LIN {X 0,Y 217.239,Z 668.067,A -85,B 0,C 180,E1 -28167.228,E2 -28167.228} C_VEL
LIN {X 0,Y 217.016,Z 676.061,A -85,B 0,C 180,E1 -28170,E2 -28170} C_VEL
LIN {X 0,Y 216.714,Z 682.608,A -85,B 0,C 180,E1 -28172.779,E2 -28172.779} C_VEL
LIN {X 0,Y 216.451,Z 688.034,A -85,B 0,C 180,E1 -28175.571,E2 -28175.571} C_VEL
LIN {X 0,Y 216.7,Z 693.898,A -85,B 0,C 180,E1 -28179.3,E2 -28179.3} C_VEL
LIN {X 0,Y 217.929,Z 698.427,A -85,B 0,C 180,E1 -28183.002,E2 -28183.002} C_VEL
LIN {X 0,Y 220.325,Z 701.768,A -85,B 0,C 180,E1 -28186.626,E2 -28186.626} C_VEL
LIN {X 0,Y 224.003,Z 703.996,A -85,B 0,C 180,E1 -28190.118,E2 -28190.118} C_VEL
LIN {X 0,Y 228.64,Z 705.109,A -85,B 0,C 180,E1 -28193.469,E2 -28193.469} C_VEL
LIN {X 0,Y 234.186,Z 705.102,A -85,B 0,C 180,E1 -28196.657,E2 -28196.657} C_VEL
LIN {X 0,Y 240.893,Z 703.976,A -85,B 0,C 180,E1 -28199.624,E2 -28199.624} C_VEL
LIN {X 0,Y 248.473,Z 701.716,A -85,B 0,C 180,E1 -28202.385,E2 -28202.385} C_VEL
LIN {X 0,Y 256.781,Z 698.288,A -85,B 0,C 180,E1 -28204.948,E2 -28204.948} C_VEL
LIN {X 0,Y 265.851,Z 693.598,A -85,B 0,C 180,E1 -28207.3,E2 -28207.3} C_VEL
LIN {X 0,Y 275.55,Z 687.57,A -85,B 0,C 180,E1 -28209.457,E2 -28209.457} C_VEL
LIN {X 0,Y 285.928,Z 680.01,A -85,B 0,C 180,E1 -28211.409,E2 -28211.409} C_VEL
LIN {X 0,Y 295.434,Z 671.975,A -85,B 0,C 180,E1 -28212.971,E2 -28212.971} C_VEL
LIN {X 0,Y 305.558,Z 662.13,A -85,B 0,C 180,E1 -28214.425,E2 -28214.425} C_VEL
LIN {X 0,Y 309.138,Z 658.314,A -85,B 0,C 180,E1 -28214.894,E2 -28214.894} C_VEL
LIN {X 0,Y 308.469,Z 659.033,A -85,B 0,C 180,E1 -28215.258,E2 -28215.258} C_VEL
LIN {X 0,Y 298.953,Z 668.646,A -85,B 0,C 180,E1 -28216.579,E2 -28216.579} C_VEL
LIN {X 0,Y 288.846,Z 677.542,A -85,B 0,C 180,E1 -28218.174,E2 -28218.174} C_VEL
LIN {X 0,Y 278.403,Z 685.481,A -85,B 0,C 180,E1 -28220.092,E2 -28220.092} C_VEL
LIN {X 0,Y 268.541,Z 691.868,A -85,B 0,C 180,E1 -28222.197,E2 -28222.197} C_VEL
LIN {X 0,Y 259.322,Z 696.857,A -85,B 0,C 180,E1 -28224.499,E2 -28224.499} C_VEL
LIN {X 0,Y 252.853,Z 699.744,A -85,B 0,C 180,E1 -28226.356,E2 -28226.356} C_VEL
LIN {X 0,Y 244.939,Z 702.551,A -85,B 0,C 180,E1 -28229.02,E2 -28229.02} C_VEL
LIN {X 0,Y 237.854,Z 704.212,A -85,B 0,C 180,E1 -28231.89,E2 -28231.89} C_VEL
LIN {X 0,Y 231.589,Z 704.754,A -85,B 0,C 180,E1 -28234.949,E2 -28234.949} C_VEL
LIN {X 0,Y 226.489,Z 704.166,A -85,B 0,C 180,E1 -28238.216,E2 -28238.216} C_VEL
LIN {X 0,Y 222.289,Z 702.473,A -85,B 0,C 180,E1 -28241.633,E2 -28241.633} C_VEL
LIN {X 0,Y 219.173,Z 699.666,A -85,B 0,C 180,E1 -28245.187,E2 -28245.187} C_VEL
LIN {X 0,Y 217.112,Z 695.687,A -85,B 0,C 180,E1 -28248.839,E2 -28248.839} C_VEL
LIN {X 0,Y 216.411,Z 690.516,A -85,B 0,C 180,E1 -28252.562,E2 -28252.562} C_VEL
LIN {X 0,Y 216.378,Z 683.877,A -85,B 0,C 180,E1 -28256.288,E2 -28256.288} C_VEL
LIN {X 0,Y 216.81,Z 676.605,A -85,B 0,C 180,E1 -28259.538,E2 -28259.538} C_VEL
LIN {X 0,Y 217.071,Z 668.937,A -85,B 0,C 180,E1 -28262.312,E2 -28262.312} C_VEL
LIN {X 0,Y 217.177,Z 661.275,A -85,B 0,C 180,E1 -28264.625,E2 -28264.625} C_VEL
LIN {X 0,Y 217.564,Z 649.405,A -85,B 0,C 180,E1 -28267.632,E2 -28267.632} C_VEL
LIN {X 0,Y 218.06,Z 637.025,A -85,B 0,C 180,E1 -28270.176,E2 -28270.176} C_VEL
LIN {X 0,Y 218.634,Z 624.743,A -85,B 0,C 180,E1 -28272.255,E2 -28272.255} C_VEL
LIN {X 0,Y 219.439,Z 609.747,A -85,B 0,C 180,E1 -28274.323,E2 -28274.323} C_VEL
LIN {X 0,Y 220.122,Z 596.007,A -85,B 0,C 180,E1 -28275.812,E2 -28275.812} C_VEL
LIN {X 0,Y 220.726,Z 579.884,A -85,B 0,C 180,E1 -28277.129,E2 -28277.129} C_VEL
LIN {X 0,Y 222.344,Z 529.839,A -85,B 0,C 180,E1 -28280.216,E2 -28280.216} C_VEL
LIN {X 0,Y 224.364,Z 480.881,A -85,B 0,C 180,E1 -28283.122,E2 -28283.122} C_VEL
LIN {X 0,Y 222.412,Z 452.386,A -85,B 0,C 180,E1 -28284.782,E2 -28284.782} C_VEL
LIN {X 0,Y 222.243,Z 439.496,A -85,B 0,C 180,E1 -28285.563,E2 -28285.563} C_VEL
LIN {X 0,Y 225.384,Z 413.949,A -85,B 0,C 180,E1 -28290.85,E2 -28290.85} C_VEL
LIN {X 0,Y 226.091,Z 408.23,A -85,B 0,C 180,E1 -28292.026,E2 -28292.026} C_VEL
LIN {X 0,Y 221.954,Z 389.076,A -85,B 0,C 180,E1 -28296.281,E2 -28296.281} C_VEL
LIN {X 0,Y 217.974,Z 370.88,A -85,B 0,C 180,E1 -28300.539,E2 -28300.539} C_VEL
LIN {X 0,Y 217.957,Z 370.883,A -85,B 0,C 180,E1 -28305.008,E2 -28305.008} C_VEL
LIN {X 0,Y 217.914,Z 370.887,A -85,B 0,C 180,E1 -28309.995,E2 -28309.995} C_VEL
LIN {X 0,Y 217.915,Z 371.065,A -85,B 0,C 180,E1 -28312.499,E2 -28312.499} C_VEL
LIN {X 0,Y 218.846,Z 373.704,A -85,B 0,C 180,E1 -28312.823,E2 -28312.823} C_VEL
LIN {X 0,Y 220.752,Z 376.135,A -85,B 0,C 180,E1 -28313.348,E2 -28313.348} C_VEL
LIN {X 0,Y 228.182,Z 388.008,A -85,B 0,C 180,E1 -28315.37,E2 -28315.37} C_VEL
LIN {X 0,Y 235.262,Z 400.411,A -85,B 0,C 180,E1 -28317.173,E2 -28317.173} C_VEL
LIN {X 0,Y 242.271,Z 414.273,A -85,B 0,C 180,E1 -28318.874,E2 -28318.874} C_VEL
LIN {X 0,Y 245.306,Z 421.27,A -85,B 0,C 180,E1 -28319.604,E2 -28319.604} C_VEL
LIN {X 0,Y 243.354,Z 467.862,A -85,B 0,C 180,E1 -28320.91,E2 -28320.91} C_VEL
LIN {X 0,Y 242.688,Z 488.569,A -85,B 0,C 180,E1 -28321.593,E2 -28321.593} C_VEL
LIN {X 0,Y 241.708,Z 502.885,A -85,B 0,C 180,E1 -28322.376,E2 -28322.376} C_VEL
LIN {X 0,Y 240.063,Z 516.937,A -85,B 0,C 180,E1 -28323.463,E2 -28323.463} C_VEL
LIN {X 0,Y 238.085,Z 529.464,A -85,B 0,C 180,E1 -28324.749,E2 -28324.749} C_VEL
LIN {X 0,Y 235.873,Z 541.665,A -85,B 0,C 180,E1 -28326.366,E2 -28326.366} C_VEL
LIN {X 0,Y 233.439,Z 552.842,A -85,B 0,C 180,E1 -28328.203,E2 -28328.203} C_VEL
LIN {X 0,Y 230.488,Z 564.111,A -85,B 0,C 180,E1 -28330.471,E2 -28330.471} C_VEL
LIN {X 0,Y 227.585,Z 574.185,A -85,B 0,C 180,E1 -28332.999,E2 -28332.999} C_VEL
LIN {X 0,Y 225.054,Z 582.522,A -85,B 0,C 180,E1 -28335.583,E2 -28335.583} C_VEL
LIN {X 0,Y 222.582,Z 590.486,A -85,B 0,C 180,E1 -28338.657,E2 -28338.657} C_VEL
LIN {X 0,Y 220.534,Z 596.925,A -85,B 0,C 180,E1 -28341.783,E2 -28341.783} C_VEL
LIN {X 0,Y 218.897,Z 602.636,A -85,B 0,C 180,E1 -28345.412,E2 -28345.412} C_VEL
LIN {X 0,Y 217.896,Z 605.963,A -85,B 0,C 180,E1 -28348.158,E2 -28348.158} C_VEL
LIN {X 0,Y 217.342,Z 609.076,A -85,B 0,C 180,E1 -28351.847,E2 -28351.847} C_VEL
LIN {X 0,Y 217.4,Z 610.861,A -85,B 0,C 180,E1 -28355.547,E2 -28355.547} C_VEL
LIN {X 0,Y 217.897,Z 611.372,A -85,B 0,C 180,E1 -28359.25,E2 -28359.25} C_VEL
LIN {X 0,Y 218.987,Z 610.594,A -85,B 0,C 180,E1 -28362.939,E2 -28362.939} C_VEL
LIN {X 0,Y 220.846,Z 608.486,A -85,B 0,C 180,E1 -28366.586,E2 -28366.586} C_VEL
LIN {X 0,Y 223.353,Z 604.998,A -85,B 0,C 180,E1 -28370.18,E2 -28370.18} C_VEL
LIN {X 0,Y 226.54,Z 600.015,A -85,B 0,C 180,E1 -28373.701,E2 -28373.701} C_VEL
LIN {X 0,Y 229.333,Z 595.158,A -85,B 0,C 180,E1 -28376.287,E2 -28376.287} C_VEL
LIN {X 0,Y 232.549,Z 589.258,A -85,B 0,C 180,E1 -28378.812,E2 -28378.812} C_VEL
LIN {X 0,Y 236.031,Z 582.148,A -85,B 0,C 180,E1 -28381.288,E2 -28381.288} C_VEL
LIN {X 0,Y 239.912,Z 573.556,A -85,B 0,C 180,E1 -28383.692,E2 -28383.692} C_VEL
LIN {X 0,Y 244.123,Z 563.102,A -85,B 0,C 180,E1 -28386.029,E2 -28386.029} C_VEL
LIN {X 0,Y 247.683,Z 552.705,A -85,B 0,C 180,E1 -28387.919,E2 -28387.919} C_VEL
LIN {X 0,Y 251.273,Z 540.922,A -85,B 0,C 180,E1 -28389.618,E2 -28389.618} C_VEL
LIN {X 0,Y 254.091,Z 529.856,A -85,B 0,C 180,E1 -28390.898,E2 -28390.898} C_VEL
LIN {X 0,Y 256.455,Z 517.32,A -85,B 0,C 180,E1 -28392.089,E2 -28392.089} C_VEL
LIN {X 0,Y 258.384,Z 503.779,A -85,B 0,C 180,E1 -28393.059,E2 -28393.059} C_VEL
LIN {X 0,Y 259.712,Z 489.587,A -85,B 0,C 180,E1 -28393.773,E2 -28393.773} C_VEL
LIN {X 0,Y 260.854,Z 465.343,A -85,B 0,C 180,E1 -28394.506,E2 -28394.506} C_VEL
LIN {X 0,Y 262.236,Z 439.318,A -85,B 0,C 180,E1 -28395.181,E2 -28395.181} C_VEL
LIN {X 0,Y 255.219,Z 425.613,A -85,B 0,C 180,E1 -28397.213,E2 -28397.213} C_VEL
LIN {X 0,Y 248.037,Z 413.291,A -85,B 0,C 180,E1 -28399.428,E2 -28399.428} C_VEL
LIN {X 0,Y 241.222,Z 402.723,A -85,B 0,C 180,E1 -28401.7,E2 -28401.7} C_VEL
LIN {X 0,Y 235.069,Z 393.963,A -85,B 0,C 180,E1 -28403.931,E2 -28403.931} C_VEL
LIN {X 0,Y 231.964,Z 389.746,A -85,B 0,C 180,E1 -28405.137,E2 -28405.137} C_VEL
LIN {X 0,Y 229.146,Z 385.959,A -85,B 0,C 180,E1 -28406.289,E2 -28406.289} C_VEL
LIN {X 0,Y 226.552,Z 382.584,A -85,B 0,C 180,E1 -28407.4,E2 -28407.4} C_VEL
LIN {X 0,Y 225.628,Z 381.365,A -85,B 0,C 180,E1 -28407.81,E2 -28407.81} C_VEL
LIN {X 0,Y 223.117,Z 378.62,A -85,B 0,C 180,E1 -28408.933,E2 -28408.933} C_VEL
LIN {X 0,Y 221.93,Z 376.426,A -85,B 0,C 180,E1 -28409.538,E2 -28409.538} C_VEL
LIN {X 0,Y 219.585,Z 374.611,A -85,B 0,C 180,E1 -28410.628,E2 -28410.628} C_VEL
LIN {X 0,Y 218.259,Z 372.275,A -85,B 0,C 180,E1 -28411.354,E2 -28411.354} C_VEL
LIN {X 0,Y 217.947,Z 370.893,A -85,B 0,C 180,E1 -28411.637,E2 -28411.637} C_VEL
LIN {X 0,Y 218.133,Z 370.862,A -85,B 0,C 180,E1 -28415.626,E2 -28415.626} C_VEL
LIN {X 0,Y 221.913,Z 388.842,A -85,B 0,C 180,E1 -28416.704,E2 -28416.704} C_VEL
LIN {X 0,Y 223.294,Z 395.329,A -85,B 0,C 180,E1 -28417.075,E2 -28417.075} C_VEL
LIN {X 0,Y 221.072,Z 474.246,A -85,B 0,C 180,E1 -28421.651,E2 -28421.651} C_VEL
LIN {X 0,Y 220.452,Z 493.196,A -85,B 0,C 180,E1 -28422.909,E2 -28422.909} C_VEL
LIN {X 0,Y 219.736,Z 509.328,A -85,B 0,C 180,E1 -28424.397,E2 -28424.397} C_VEL
LIN {X 0,Y 218.934,Z 523.797,A -85,B 0,C 180,E1 -28426.116,E2 -28426.116} C_VEL
LIN {X 0,Y 218.262,Z 537.78,A -85,B 0,C 180,E1 -28428.194,E2 -28428.194} C_VEL
LIN {X 0,Y 217.565,Z 550.552,A -85,B 0,C 180,E1 -28430.502,E2 -28430.502} C_VEL
LIN {X 0,Y 217.002,Z 562.308,A -85,B 0,C 180,E1 -28433.047,E2 -28433.047} C_VEL
LIN {X 0,Y 216.744,Z 573.124,A -85,B 0,C 180,E1 -28435.83,E2 -28435.83} C_VEL
LIN {X 0,Y 216.798,Z 582.245,A -85,B 0,C 180,E1 -28438.611,E2 -28438.611} C_VEL
LIN {X 0,Y 217.104,Z 591.161,A -85,B 0,C 180,E1 -28441.848,E2 -28441.848} C_VEL
LIN {X 0,Y 218.282,Z 599.669,A -85,B 0,C 180,E1 -28445.524,E2 -28445.524} C_VEL
LIN {X 0,Y 220.437,Z 606.463,A -85,B 0,C 180,E1 -28449.141,E2 -28449.141} C_VEL
LIN {X 0,Y 223.32,Z 611.825,A -85,B 0,C 180,E1 -28452.682,E2 -28452.682} C_VEL
LIN {X 0,Y 227.183,Z 615.845,A -85,B 0,C 180,E1 -28456.11,E2 -28456.11} C_VEL
LIN {X 0,Y 232.285,Z 618.601,A -85,B 0,C 180,E1 -28459.372,E2 -28459.372} C_VEL
LIN {X 0,Y 238.281,Z 620.078,A -85,B 0,C 180,E1 -28462.466,E2 -28462.466} C_VEL
LIN {X 0,Y 244.834,Z 620.332,A -85,B 0,C 180,E1 -28465.412,E2 -28465.412} C_VEL
LIN {X 0,Y 252.123,Z 619.353,A -85,B 0,C 180,E1 -28468.183,E2 -28468.183} C_VEL
LIN {X 0,Y 260.145,Z 617.068,A -85,B 0,C 180,E1 -28470.769,E2 -28470.769} C_VEL
LIN {X 0,Y 268.722,Z 613.52,A -85,B 0,C 180,E1 -28473.187,E2 -28473.187} C_VEL
LIN {X 0,Y 277.79,Z 608.573,A -85,B 0,C 180,E1 -28475.446,E2 -28475.446} C_VEL
LIN {X 0,Y 284.981,Z 603.815,A -85,B 0,C 180,E1 -28477.026,E2 -28477.026} C_VEL
LIN {X 0,Y 291.336,Z 598.971,A -85,B 0,C 180,E1 -28478.322,E2 -28478.322} C_VEL
LIN {X 0,Y 293.48,Z 597.269,A -85,B 0,C 180,E1 -28478.892,E2 -28478.892} C_VEL
LIN {X 0,Y 298.813,Z 592.901,A -85,B 0,C 180,E1 -28481.142,E2 -28481.142} C_VEL
LIN {X 0,Y 301.043,Z 590.943,A -85,B 0,C 180,E1 -28481.645,E2 -28481.645} C_VEL
LIN {X 0,Y 305.429,Z 586.722,A -85,B 0,C 180,E1 -28482.335,E2 -28482.335} C_VEL
LIN {X 0,Y 304.596,Z 587.747,A -85,B 0,C 180,E1 -28482.619,E2 -28482.619} C_VEL
LIN {X 0,Y 294.305,Z 598.624,A -85,B 0,C 180,E1 -28483.785,E2 -28483.785} C_VEL
LIN {X 0,Y 283.48,Z 608.692,A -85,B 0,C 180,E1 -28485.235,E2 -28485.235} C_VEL
LIN {X 0,Y 272.282,Z 617.864,A -85,B 0,C 180,E1 -28487.022,E2 -28487.022} C_VEL
LIN {X 0,Y 261.742,Z 625.352,A -85,B 0,C 180,E1 -28489.031,E2 -28489.031} C_VEL
LIN {X 0,Y 252.03,Z 631.45,A -85,B 0,C 180,E1 -28491.294,E2 -28491.294} C_VEL
LIN {X 0,Y 241.938,Z 636.847,A -85,B 0,C 180,E1 -28494.158,E2 -28494.158} C_VEL
LIN {X 0,Y 233.229,Z 640.723,A -85,B 0,C 180,E1 -28497.276,E2 -28497.276} C_VEL
LIN {X 0,Y 226.564,Z 643.134,A -85,B 0,C 180,E1 -28500.352,E2 -28500.352} C_VEL
LIN {X 0,Y 220.828,Z 644.503,A -85,B 0,C 180,E1 -28503.636,E2 -28503.636} C_VEL
LIN {X 0,Y 216.414,Z 644.876,A -85,B 0,C 180,E1 -28507.145,E2 -28507.145} C_VEL
LIN {X 0,Y 213.801,Z 644.649,A -85,B 0,C 180,E1 -28510.129,E2 -28510.129} C_VEL
LIN {X 0,Y 211.059,Z 649.675,A -85,B 0,C 180,E1 -28513.615,E2 -28513.615} C_VEL
LIN {X 0,Y 209.681,Z 652.77,A -85,B 0,C 180,E1 -28516.477,E2 -28516.477} C_VEL
LIN {X 0,Y 209.155,Z 655.731,A -85,B 0,C 180,E1 -28520.36,E2 -28520.36} C_VEL
LIN {X 0,Y 210.103,Z 657.418,A -85,B 0,C 180,E1 -28524.26,E2 -28524.26} C_VEL
LIN {X 0,Y 210.454,Z 657.715,A -85,B 0,C 180,E1 -28525.047,E2 -28525.047} C_VEL
LIN {X 0,Y 210.457,Z 666.558,A -85,B 0,C 180,E1 -28527.615,E2 -28527.615} C_VEL
LIN {X 0,Y 210.243,Z 675.083,A -85,B 0,C 180,E1 -28530.621,E2 -28530.621} C_VEL
LIN {X 0,Y 209.973,Z 680.381,A -85,B 0,C 180,E1 -28532.868,E2 -28532.868} C_VEL
LIN {X 0,Y 209.631,Z 687.756,A -85,B 0,C 180,E1 -28536.716,E2 -28536.716} C_VEL
LIN {X 0,Y 210.001,Z 693.577,A -85,B 0,C 180,E1 -28540.57,E2 -28540.57} C_VEL
LIN {X 0,Y 211.145,Z 697.115,A -85,B 0,C 180,E1 -28543.427,E2 -28543.427} C_VEL
LIN {X 0,Y 213.61,Z 700.776,A -85,B 0,C 180,E1 -28547.164,E2 -28547.164} C_VEL
LIN {X 0,Y 217.376,Z 703.337,A -85,B 0,C 180,E1 -28550.759,E2 -28550.759} C_VEL
LIN {X 0,Y 222.146,Z 704.799,A -85,B 0,C 180,E1 -28554.198,E2 -28554.198} C_VEL
LIN {X 0,Y 227.875,Z 705.189,A -85,B 0,C 180,E1 -28557.456,E2 -28557.456} C_VEL
LIN {X 0,Y 234.778,Z 704.493,A -85,B 0,C 180,E1 -28560.476,E2 -28560.476} C_VEL
LIN {X 0,Y 242.563,Z 702.672,A -85,B 0,C 180,E1 -28563.275,E2 -28563.275} C_VEL
LIN {X 0,Y 251.087,Z 699.702,A -85,B 0,C 180,E1 -28565.861,E2 -28565.861} C_VEL
LIN {X 0,Y 260.361,Z 695.524,A -85,B 0,C 180,E1 -28568.226,E2 -28568.226} C_VEL
LIN {X 0,Y 270.302,Z 690.053,A -85,B 0,C 180,E1 -28570.378,E2 -28570.378} C_VEL
LIN {X 0,Y 280.858,Z 683.145,A -85,B 0,C 180,E1 -28572.327,E2 -28572.327} C_VEL
LIN {X 0,Y 291.986,Z 674.556,A -85,B 0,C 180,E1 -28574.081,E2 -28574.081} C_VEL
LIN {X 0,Y 297.725,Z 669.572,A -85,B 0,C 180,E1 -28574.894,E2 -28574.894} C_VEL
LIN {X 0,Y 297.968,Z 669.35,A -85,B 0,C 180,E1 -28575.153,E2 -28575.153} C_VEL
LIN {X 0,Y 286.626,Z 678.812,A -85,B 0,C 180,E1 -28576.824,E2 -28576.824} C_VEL
LIN {X 0,Y 275.847,Z 686.49,A -85,B 0,C 180,E1 -28578.685,E2 -28578.685} C_VEL
LIN {X 0,Y 265.582,Z 692.649,A -85,B 0,C 180,E1 -28580.73,E2 -28580.73} C_VEL
LIN {X 0,Y 255.965,Z 697.438,A -85,B 0,C 180,E1 -28582.985,E2 -28582.985} C_VEL
LIN {X 0,Y 247.049,Z 700.974,A -85,B 0,C 180,E1 -28585.456,E2 -28585.456} C_VEL
LIN {X 0,Y 238.93,Z 703.324,A -85,B 0,C 180,E1 -28588.151,E2 -28588.151} C_VEL
LIN {X 0,Y 231.634,Z 704.547,A -85,B 0,C 180,E1 -28591.065,E2 -28591.065} C_VEL
LIN {X 0,Y 225.194,Z 704.676,A -85,B 0,C 180,E1 -28594.186,E2 -28594.186} C_VEL
LIN {X 0,Y 219.932,Z 703.729,A -85,B 0,C 180,E1 -28597.532,E2 -28597.532} C_VEL
LIN {X 0,Y 215.6,Z 701.701,A -85,B 0,C 180,E1 -28601.042,E2 -28601.042} C_VEL
LIN {X 0,Y 212.393,Z 698.565,A -85,B 0,C 180,E1 -28604.703,E2 -28604.703} C_VEL
LIN {X 0,Y 210.303,Z 694.256,A -85,B 0,C 180,E1 -28608.473,E2 -28608.473} C_VEL
LIN {X 0,Y 209.61,Z 688.753,A -85,B 0,C 180,E1 -28612.319,E2 -28612.319} C_VEL
LIN {X 0,Y 209.619,Z 681.739,A -85,B 0,C 180,E1 -28616.169,E2 -28616.169} C_VEL
LIN {X 0,Y 210,Z 675.356,A -85,B 0,C 180,E1 -28619.045,E2 -28619.045} C_VEL
LIN {X 0,Y 210.293,Z 667.543,A -85,B 0,C 180,E1 -28621.909,E2 -28621.909} C_VEL
LIN {X 0,Y 210.372,Z 659.723,A -85,B 0,C 180,E1 -28624.297,E2 -28624.297} C_VEL
LIN {X 0,Y 210.702,Z 648.606,A -85,B 0,C 180,E1 -28627.162,E2 -28627.162} C_VEL
LIN {X 0,Y 211.158,Z 636.133,A -85,B 0,C 180,E1 -28629.789,E2 -28629.789} C_VEL
LIN {X 0,Y 211.705,Z 623.81,A -85,B 0,C 180,E1 -28631.935,E2 -28631.935} C_VEL
LIN {X 0,Y 212.407,Z 610.481,A -85,B 0,C 180,E1 -28633.833,E2 -28633.833} C_VEL
LIN {X 0,Y 213.124,Z 595.883,A -85,B 0,C 180,E1 -28635.488,E2 -28635.488} C_VEL
LIN {X 0,Y 213.702,Z 579.916,A -85,B 0,C 180,E1 -28636.851,E2 -28636.851} C_VEL
LIN {X 0,Y 215.13,Z 534.137,A -85,B 0,C 180,E1 -28639.805,E2 -28639.805} C_VEL
LIN {X 0,Y 217.198,Z 480.47,A -85,B 0,C 180,E1 -28643.133,E2 -28643.133} C_VEL
LIN {X 0,Y 215.308,Z 451.499,A -85,B 0,C 180,E1 -28644.879,E2 -28644.879} C_VEL
LIN {X 0,Y 215.154,Z 439.583,A -85,B 0,C 180,E1 -28645.619,E2 -28645.619} C_VEL
LIN {X 0,Y 218.397,Z 413.625,A -85,B 0,C 180,E1 -28651.143,E2 -28651.143} C_VEL
LIN {X 0,Y 218.981,Z 408.973,A -85,B 0,C 180,E1 -28652.126,E2 -28652.126} C_VEL
LIN {X 0,Y 214.438,Z 387.924,A -85,B 0,C 180,E1 -28656.918,E2 -28656.918} C_VEL
LIN {X 0,Y 210.918,Z 371.757,A -85,B 0,C 180,E1 -28660.775,E2 -28660.775} C_VEL
LIN {X 0,Y 210.867,Z 371.765,A -85,B 0,C 180,E1 -28665.768,E2 -28665.768} C_VEL
LIN {X 0,Y 210.869,Z 371.769,A -85,B 0,C 180,E1 -28670.818,E2 -28670.818} C_VEL
LIN {X 0,Y 211.871,Z 374.667,A -85,B 0,C 180,E1 -28671.226,E2 -28671.226} C_VEL
LIN {X 0,Y 213.861,Z 377.191,A -85,B 0,C 180,E1 -28671.819,E2 -28671.819} C_VEL
LIN {X 0,Y 216.064,Z 380.489,A -85,B 0,C 180,E1 -28672.48,E2 -28672.48} C_VEL
LIN {X 0,Y 223.922,Z 393.095,A -85,B 0,C 180,E1 -28674.715,E2 -28674.715} C_VEL
LIN {X 0,Y 231.595,Z 406.867,A -85,B 0,C 180,E1 -28676.748,E2 -28676.748} C_VEL
LIN {X 0,Y 238.341,Z 420.942,A -85,B 0,C 180,E1 -28678.46,E2 -28678.46} C_VEL
LIN {X 0,Y 239.293,Z 423.137,A -85,B 0,C 180,E1 -28678.698,E2 -28678.698} C_VEL
LIN {X 0,Y 237.334,Z 470.751,A -85,B 0,C 180,E1 -28680.078,E2 -28680.078} C_VEL
LIN {X 0,Y 236.679,Z 489.602,A -85,B 0,C 180,E1 -28680.725,E2 -28680.725} C_VEL
LIN {X 0,Y 235.58,Z 504.115,A -85,B 0,C 180,E1 -28681.537,E2 -28681.537} C_VEL
LIN {X 0,Y 233.968,Z 517.449,A -85,B 0,C 180,E1 -28682.594,E2 -28682.594} C_VEL
LIN {X 0,Y 231.763,Z 530.898,A -85,B 0,C 180,E1 -28684.009,E2 -28684.009} C_VEL
LIN {X 0,Y 229.482,Z 542.965,A -85,B 0,C 180,E1 -28685.666,E2 -28685.666} C_VEL
LIN {X 0,Y 226.939,Z 554.05,A -85,B 0,C 180,E1 -28687.545,E2 -28687.545} C_VEL
LIN {X 0,Y 223.88,Z 565.239,A -85,B 0,C 180,E1 -28689.87,E2 -28689.87} C_VEL
LIN {X 0,Y 220.861,Z 575.233,A -85,B 0,C 180,E1 -28692.465,E2 -28692.465} C_VEL
LIN {X 0,Y 218.256,Z 583.522,A -85,B 0,C 180,E1 -28695.123,E2 -28695.123} C_VEL
LIN {X 0,Y 215.698,Z 591.44,A -85,B 0,C 180,E1 -28698.29,E2 -28698.29} C_VEL
LIN {X 0,Y 213.582,Z 597.841,A -85,B 0,C 180,E1 -28701.514,E2 -28701.514} C_VEL
LIN {X 0,Y 211.874,Z 603.52,A -85,B 0,C 180,E1 -28705.259,E2 -28705.259} C_VEL
LIN {X 0,Y 210.842,Z 606.815,A -85,B 0,C 180,E1 -28708.097,E2 -28708.097} C_VEL
LIN {X 0,Y 210.28,Z 610.02,A -85,B 0,C 180,E1 -28712.121,E2 -28712.121} C_VEL
LIN {X 0,Y 210.356,Z 611.653,A -85,B 0,C 180,E1 -28715.733,E2 -28715.733} C_VEL
LIN {X 0,Y 210.893,Z 612.136,A -85,B 0,C 180,E1 -28719.56,E2 -28719.56} C_VEL
LIN {X 0,Y 212.061,Z 611.328,A -85,B 0,C 180,E1 -28723.369,E2 -28723.369} C_VEL
LIN {X 0,Y 214.05,Z 609.188,A -85,B 0,C 180,E1 -28727.129,E2 -28727.129} C_VEL
LIN {X 0,Y 216.708,Z 605.668,A -85,B 0,C 180,E1 -28730.827,E2 -28730.827} C_VEL
LIN {X 0,Y 220.051,Z 600.651,A -85,B 0,C 180,E1 -28734.444,E2 -28734.444} C_VEL
LIN {X 0,Y 222.986,Z 595.756,A -85,B 0,C 180,E1 -28737.096,E2 -28737.096} C_VEL
LIN {X 0,Y 226.329,Z 589.818,A -85,B 0,C 180,E1 -28739.681,E2 -28739.681} C_VEL
LIN {X 0,Y 230.623,Z 581.327,A -85,B 0,C 180,E1 -28742.623,E2 -28742.623} C_VEL
LIN {X 0,Y 234.789,Z 572.404,A -85,B 0,C 180,E1 -28745.05,E2 -28745.05} C_VEL
LIN {X 0,Y 239.1,Z 561.572,A -85,B 0,C 180,E1 -28747.436,E2 -28747.436} C_VEL
LIN {X 0,Y 242.987,Z 550.495,A -85,B 0,C 180,E1 -28749.36,E2 -28749.36} C_VEL
LIN {X 0,Y 246.72,Z 538.193,A -85,B 0,C 180,E1 -28751.036,E2 -28751.036} C_VEL
LIN {X 0,Y 249.473,Z 526.301,A -85,B 0,C 180,E1 -28752.365,E2 -28752.365} C_VEL
LIN {X 0,Y 251.996,Z 512.17,A -85,B 0,C 180,E1 -28753.578,E2 -28753.578} C_VEL
LIN {X 0,Y 253.754,Z 498.145,A -85,B 0,C 180,E1 -28754.456,E2 -28754.456} C_VEL
LIN {X 0,Y 254.81,Z 483.931,A -85,B 0,C 180,E1 -28755.047,E2 -28755.047} C_VEL
LIN {X 0,Y 256.902,Z 441.691,A -85,B 0,C 180,E1 -28756.217,E2 -28756.217} C_VEL
LIN {X 0,Y 249.611,Z 427.57,A -85,B 0,C 180,E1 -28758.448,E2 -28758.448} C_VEL
LIN {X 0,Y 242.071,Z 414.777,A -85,B 0,C 180,E1 -28760.926,E2 -28760.926} C_VEL
LIN {X 0,Y 235.107,Z 404.149,A -85,B 0,C 180,E1 -28763.426,E2 -28763.426} C_VEL
LIN {X 0,Y 229.288,Z 395.913,A -85,B 0,C 180,E1 -28765.719,E2 -28765.719} C_VEL
LIN {X 0,Y 226.11,Z 391.679,A -85,B 0,C 180,E1 -28767.064,E2 -28767.064} C_VEL
LIN {X 0,Y 222.747,Z 387.275,A -85,B 0,C 180,E1 -28768.579,E2 -28768.579} C_VEL
LIN {X 0,Y 220.121,Z 384.057,A -85,B 0,C 180,E1 -28769.826,E2 -28769.826} C_VEL
LIN {X 0,Y 219.258,Z 382.674,A -85,B 0,C 180,E1 -28770.272,E2 -28770.272} C_VEL
LIN {X 0,Y 216.637,Z 380.105,A -85,B 0,C 180,E1 -28771.582,E2 -28771.582} C_VEL
LIN {X 0,Y 215.079,Z 377.381,A -85,B 0,C 180,E1 -28772.48,E2 -28772.48} C_VEL
LIN {X 0,Y 212.683,Z 375.598,A -85,B 0,C 180,E1 -28773.771,E2 -28773.771} C_VEL
LIN {X 0,Y 211.373,Z 373.252,A -85,B 0,C 180,E1 -28774.613,E2 -28774.613} C_VEL
LIN {X 0,Y 211.034,Z 371.739,A -85,B 0,C 180,E1 -28774.964,E2 -28774.964} C_VEL
LIN {X 0,Y 211.103,Z 371.818,A -85,B 0,C 180,E1 -28775.668,E2 -28775.668} C_VEL
LIN {X 0,Y 214.707,Z 389.117,A -85,B 0,C 180,E1 -28776.709,E2 -28776.709} C_VEL
LIN {X 0,Y 216.167,Z 396.048,A -85,B 0,C 180,E1 -28777.117,E2 -28777.117} C_VEL
LIN {X 0,Y 214.032,Z 474.095,A -85,B 0,C 180,E1 -28781.842,E2 -28781.842} C_VEL
LIN {X 0,Y 213.386,Z 493.735,A -85,B 0,C 180,E1 -28783.185,E2 -28783.185} C_VEL
LIN {X 0,Y 212.641,Z 509.697,A -85,B 0,C 180,E1 -28784.72,E2 -28784.72} C_VEL
LIN {X 0,Y 211.828,Z 524.97,A -85,B 0,C 180,E1 -28786.616,E2 -28786.616} C_VEL
LIN {X 0,Y 211.179,Z 538.86,A -85,B 0,C 180,E1 -28788.763,E2 -28788.763} C_VEL
LIN {X 0,Y 210.49,Z 551.58,A -85,B 0,C 180,E1 -28791.146,E2 -28791.146} C_VEL
LIN {X 0,Y 209.962,Z 563.284,A -85,B 0,C 180,E1 -28793.775,E2 -28793.775} C_VEL
LIN {X 0,Y 209.81,Z 573.964,A -85,B 0,C 180,E1 -28796.65,E2 -28796.65} C_VEL
LIN {X 0,Y 209.905,Z 583.048,A -85,B 0,C 180,E1 -28799.522,E2 -28799.522} C_VEL
LIN {X 0,Y 210.351,Z 592.014,A -85,B 0,C 180,E1 -28802.863,E2 -28802.863} C_VEL
LIN {X 0,Y 211.755,Z 600.442,A -85,B 0,C 180,E1 -28806.648,E2 -28806.648} C_VEL
LIN {X 0,Y 214.117,Z 607.333,A -85,B 0,C 180,E1 -28810.365,E2 -28810.365} C_VEL
LIN {X 0,Y 217.303,Z 612.72,A -85,B 0,C 180,E1 -28813.989,E2 -28813.989} C_VEL
LIN {X 0,Y 220.393,Z 615.909,A -85,B 0,C 180,E1 -28816.62,E2 -28816.62} C_VEL
LIN {X 0,Y 225.619,Z 619.062,A -85,B 0,C 180,E1 -28819.968,E2 -28819.968} C_VEL
LIN {X 0,Y 231.77,Z 620.958,A -85,B 0,C 180,E1 -28823.133,E2 -28823.133} C_VEL
LIN {X 0,Y 238.551,Z 621.628,A -85,B 0,C 180,E1 -28826.131,E2 -28826.131} C_VEL
LIN {X 0,Y 246.044,Z 621.076,A -85,B 0,C 180,E1 -28828.944,E2 -28828.944} C_VEL
LIN {X 0,Y 254.312,Z 619.267,A -85,B 0,C 180,E1 -28831.554,E2 -28831.554} C_VEL
LIN {X 0,Y 263.121,Z 616.163,A -85,B 0,C 180,E1 -28833.989,E2 -28833.989} C_VEL
LIN {X 0,Y 272.448,Z 611.737,A -85,B 0,C 180,E1 -28836.25,E2 -28836.25} C_VEL
LIN {X 0,Y 282.333,Z 605.766,A -85,B 0,C 180,E1 -28838.333,E2 -28838.333} C_VEL
LIN {X 0,Y 291.355,Z 599.236,A -85,B 0,C 180,E1 -28840.023,E2 -28840.023} C_VEL
LIN {X 0,Y 301.043,Z 590.943,A -85,B 0,C 180,E1 -28841.645,E2 -28841.645} C_VEL
LIN {X 0,Y 301.08,Z 591.024,A -85,B 0,C 180,E1 -28841.862,E2 -28841.862} C_VEL
LIN {X 0,Y 299.998,Z 592.236,A -85,B 0,C 180,E1 -28842.137,E2 -28842.137} C_VEL
LIN {X 0,Y 297.367,Z 594.912,A -85,B 0,C 180,E1 -28842.425,E2 -28842.425} C_VEL
LIN {X 0,Y 289.249,Z 602.328,A -85,B 0,C 180,E1 -28842.884,E2 -28842.884} C_VEL
LIN {X 0,Y 286.605,Z 604.59,A -85,B 0,C 180,E1 -28843.143,E2 -28843.143} C_VEL
LIN {X 0,Y 275.64,Z 613.557,A -85,B 0,C 180,E1 -28844.64,E2 -28844.64} C_VEL
LIN {X 0,Y 267.165,Z 619.686,A -85,B 0,C 180,E1 -28845.991,E2 -28845.991} C_VEL
LIN {X 0,Y 256.463,Z 626.594,A -85,B 0,C 180,E1 -28847.999,E2 -28847.999} C_VEL
LIN {X 0,Y 246.544,Z 632.131,A -85,B 0,C 180,E1 -28850.265,E2 -28850.265} C_VEL
LIN {X 0,Y 238.626,Z 635.926,A -85,B 0,C 180,E1 -28852.423,E2 -28852.423} C_VEL
LIN {X 0,Y 231.187,Z 639.034,A -85,B 0,C 180,E1 -28854.854,E2 -28854.854} C_VEL
LIN {X 0,Y 223.729,Z 641.535,A -85,B 0,C 180,E1 -28857.843,E2 -28857.843} C_VEL
LIN {X 0,Y 217.292,Z 643.003,A -85,B 0,C 180,E1 -28861.083,E2 -28861.083} C_VEL
LIN {X 0,Y 212.05,Z 643.513,A -85,B 0,C 180,E1 -28864.569,E2 -28864.569} C_VEL
LIN {X 0,Y 207.727,Z 643.034,A -85,B 0,C 180,E1 -28868.876,E2 -28868.876} C_VEL
LIN {X 0,Y 204.911,Z 647.784,A -85,B 0,C 180,E1 -28872.082,E2 -28872.082} C_VEL
LIN {X 0,Y 202.734,Z 652.066,A -85,B 0,C 180,E1 -28876.004,E2 -28876.004} C_VEL
LIN {X 0,Y 202.074,Z 654.996,A -85,B 0,C 180,E1 -28880.019,E2 -28880.019} C_VEL
LIN {X 0,Y 202.939,Z 656.652,A -85,B 0,C 180,E1 -28884.056,E2 -28884.056} C_VEL
LIN {X 0,Y 203.708,Z 657.019,A -85,B 0,C 180,E1 -28885.673,E2 -28885.673} C_VEL
LIN {X 0,Y 203.71,Z 664.99,A -85,B 0,C 180,E1 -28888.029,E2 -28888.029} C_VEL
LIN {X 0,Y 203.518,Z 673.277,A -85,B 0,C 180,E1 -28890.986,E2 -28890.986} C_VEL
LIN {X 0,Y 203.108,Z 680.094,A -85,B 0,C 180,E1 -28893.955,E2 -28893.955} C_VEL
LIN {X 0,Y 202.911,Z 687.403,A -85,B 0,C 180,E1 -28897.936,E2 -28897.936} C_VEL
LIN {X 0,Y 203.504,Z 693.206,A -85,B 0,C 180,E1 -28901.918,E2 -28901.918} C_VEL
LIN {X 0,Y 205.505,Z 697.82,A -85,B 0,C 180,E1 -28905.823,E2 -28905.823} C_VEL
LIN {X 0,Y 208.792,Z 701.284,A -85,B 0,C 180,E1 -28909.601,E2 -28909.601} C_VEL
LIN {X 0,Y 213.179,Z 703.623,A -85,B 0,C 180,E1 -28913.221,E2 -28913.221} C_VEL
LIN {X 0,Y 218.485,Z 704.888,A -85,B 0,C 180,E1 -28916.668,E2 -28916.668} C_VEL
LIN {X 0,Y 225.014,Z 705.119,A -85,B 0,C 180,E1 -28919.872,E2 -28919.872} C_VEL
LIN {X 0,Y 232.597,Z 704.275,A -85,B 0,C 180,E1 -28922.823,E2 -28922.823} C_VEL
LIN {X 0,Y 241.435,Z 702.2,A -85,B 0,C 180,E1 -28925.676,E2 -28925.676} C_VEL
LIN {X 0,Y 250.082,Z 699.277,A -85,B 0,C 180,E1 -28928.038,E2 -28928.038} C_VEL
LIN {X 0,Y 259.957,Z 694.982,A -85,B 0,C 180,E1 -28930.291,E2 -28930.291} C_VEL
LIN {X 0,Y 270.408,Z 689.396,A -85,B 0,C 180,E1 -28932.336,E2 -28932.336} C_VEL
LIN {X 0,Y 281.452,Z 682.352,A -85,B 0,C 180,E1 -28934.173,E2 -28934.173} C_VEL
LIN {X 0,Y 287.18,Z 678.208,A -85,B 0,C 180,E1 -28935.017,E2 -28935.017} C_VEL
LIN {X 0,Y 284.488,Z 680.209,A -85,B 0,C 180,E1 -28935.475,E2 -28935.475} C_VEL
LIN {X 0,Y 273.455,Z 687.507,A -85,B 0,C 180,E1 -28937.251,E2 -28937.251} C_VEL
LIN {X 0,Y 262.819,Z 693.43,A -85,B 0,C 180,E1 -28939.236,E2 -28939.236} C_VEL
LIN {X 0,Y 255.28,Z 696.99,A -85,B 0,C 180,E1 -28940.871,E2 -28940.871} C_VEL
LIN {X 0,Y 245.765,Z 700.638,A -85,B 0,C 180,E1 -28943.237,E2 -28943.237} C_VEL
LIN {X 0,Y 236.574,Z 703.215,A -85,B 0,C 180,E1 -28945.998,E2 -28945.998} C_VEL
LIN {X 0,Y 229.09,Z 704.463,A -85,B 0,C 180,E1 -28948.683,E2 -28948.683} C_VEL
LIN {X 0,Y 221.995,Z 704.747,A -85,B 0,C 180,E1 -28951.753,E2 -28951.753} C_VEL
LIN {X 0,Y 215.996,Z 703.971,A -85,B 0,C 180,E1 -28955.067,E2 -28955.067} C_VEL
LIN {X 0,Y 211.094,Z 702.149,A -85,B 0,C 180,E1 -28958.593,E2 -28958.593} C_VEL
LIN {X 0,Y 207.1,Z 699.204,A -85,B 0,C 180,E1 -28962.279,E2 -28962.279} C_VEL
LIN {X 0,Y 204.48,Z 695.157,A -85,B 0,C 180,E1 -28966.127,E2 -28966.127} C_VEL
LIN {X 0,Y 203.055,Z 689.918,A -85,B 0,C 180,E1 -28970.069,E2 -28970.069} C_VEL
LIN {X 0,Y 202.767,Z 685.129,A -85,B 0,C 180,E1 -28973.056,E2 -28973.056} C_VEL
LIN {X 0,Y 203.053,Z 677.362,A -85,B 0,C 180,E1 -28977.035,E2 -28977.035} C_VEL
LIN {X 0,Y 203.367,Z 670.14,A -85,B 0,C 180,E1 -28980.001,E2 -28980.001} C_VEL
LIN {X 0,Y 203.543,Z 663.151,A -85,B 0,C 180,E1 -28982.416,E2 -28982.416} C_VEL
LIN {X 0,Y 203.629,Z 654.451,A -85,B 0,C 180,E1 -28984.934,E2 -28984.934} C_VEL
LIN {X 0,Y 203.944,Z 644.503,A -85,B 0,C 180,E1 -28987.4,E2 -28987.4} C_VEL
LIN {X 0,Y 204.442,Z 632.651,A -85,B 0,C 180,E1 -28989.864,E2 -28989.864} C_VEL
LIN {X 0,Y 204.937,Z 619.543,A -85,B 0,C 180,E1 -28992.084,E2 -28992.084} C_VEL
LIN {X 0,Y 205.722,Z 605.39,A -85,B 0,C 180,E1 -28994.04,E2 -28994.04} C_VEL
LIN {X 0,Y 206.314,Z 590.707,A -85,B 0,C 180,E1 -28995.634,E2 -28995.634} C_VEL
LIN {X 0,Y 206.962,Z 573.874,A -85,B 0,C 180,E1 -28996.973,E2 -28996.973} C_VEL
LIN {X 0,Y 210.11,Z 480.59,A -85,B 0,C 180,E1 -29003.094,E2 -29003.094} C_VEL
LIN {X 0,Y 208.193,Z 451.16,A -85,B 0,C 180,E1 -29004.937,E2 -29004.937} C_VEL
LIN {X 0,Y 208.072,Z 439.493,A -85,B 0,C 180,E1 -29005.702,E2 -29005.702} C_VEL
LIN {X 0,Y 211.398,Z 413.186,A -85,B 0,C 180,E1 -29011.457,E2 -29011.457} C_VEL
LIN {X 0,Y 211.851,Z 409.714,A -85,B 0,C 180,E1 -29012.209,E2 -29012.209} C_VEL
LIN {X 0,Y 207.842,Z 390.855,A -85,B 0,C 180,E1 -29016.602,E2 -29016.602} C_VEL
LIN {X 0,Y 203.898,Z 372.632,A -85,B 0,C 180,E1 -29021.059,E2 -29021.059} C_VEL
LIN {X 0,Y 203.803,Z 372.646,A -85,B 0,C 180,E1 -29026.2,E2 -29026.2} C_VEL
LIN {X 0,Y 203.793,Z 372.648,A -85,B 0,C 180,E1 -29029.001,E2 -29029.001} C_VEL
LIN {X 0,Y 204.778,Z 375.462,A -85,B 0,C 180,E1 -29029.434,E2 -29029.434} C_VEL
LIN {X 0,Y 206.85,Z 377.945,A -85,B 0,C 180,E1 -29030.103,E2 -29030.103} C_VEL
LIN {X 0,Y 209.103,Z 381.415,A -85,B 0,C 180,E1 -29030.842,E2 -29030.842} C_VEL
LIN {X 0,Y 215.705,Z 391.572,A -85,B 0,C 180,E1 -29032.875,E2 -29032.875} C_VEL
LIN {X 0,Y 223.688,Z 405.28,A -85,B 0,C 180,E1 -29035.158,E2 -29035.158} C_VEL
LIN {X 0,Y 230.787,Z 419.376,A -85,B 0,C 180,E1 -29037.074,E2 -29037.074} C_VEL
LIN {X 0,Y 233.383,Z 425.217,A -85,B 0,C 180,E1 -29037.76,E2 -29037.76} C_VEL
LIN {X 0,Y 231.372,Z 473.091,A -85,B 0,C 180,E1 -29039.184,E2 -29039.184} C_VEL
LIN {X 0,Y 230.712,Z 490.611,A -85,B 0,C 180,E1 -29039.807,E2 -29039.807} C_VEL
LIN {X 0,Y 229.527,Z 505.309,A -85,B 0,C 180,E1 -29040.654,E2 -29040.654} C_VEL
LIN {X 0,Y 227.779,Z 519.068,A -85,B 0,C 180,E1 -29041.784,E2 -29041.784} C_VEL
LIN {X 0,Y 225.478,Z 532.332,A -85,B 0,C 180,E1 -29043.228,E2 -29043.228} C_VEL
LIN {X 0,Y 223.131,Z 544.265,A -85,B 0,C 180,E1 -29044.926,E2 -29044.926} C_VEL
LIN {X 0,Y 220.198,Z 556.361,A -85,B 0,C 180,E1 -29047.066,E2 -29047.066} C_VEL
LIN {X 0,Y 217.29,Z 566.355,A -85,B 0,C 180,E1 -29049.232,E2 -29049.232} C_VEL
LIN {X 0,Y 214.181,Z 576.277,A -85,B 0,C 180,E1 -29051.9,E2 -29051.9} C_VEL
LIN {X 0,Y 211.473,Z 584.519,A -85,B 0,C 180,E1 -29054.635,E2 -29054.635} C_VEL
LIN {X 0,Y 209.188,Z 591.394,A -85,B 0,C 180,E1 -29057.429,E2 -29057.429} C_VEL
LIN {X 0,Y 207.159,Z 597.093,A -85,B 0,C 180,E1 -29060.267,E2 -29060.267} C_VEL
LIN {X 0,Y 205.225,Z 603.176,A -85,B 0,C 180,E1 -29064.123,E2 -29064.123} C_VEL
LIN {X 0,Y 203.79,Z 607.666,A -85,B 0,C 180,E1 -29068.031,E2 -29068.031} C_VEL
LIN {X 0,Y 203.252,Z 610.714,A -85,B 0,C 180,E1 -29071.975,E2 -29071.975} C_VEL
LIN {X 0,Y 203.333,Z 612.442,A -85,B 0,C 180,E1 -29075.932,E2 -29075.932} C_VEL
LIN {X 0,Y 203.903,Z 612.898,A -85,B 0,C 180,E1 -29079.89,E2 -29079.89} C_VEL
LIN {X 0,Y 205.151,Z 612.062,A -85,B 0,C 180,E1 -29083.828,E2 -29083.828} C_VEL
LIN {X 0,Y 207.278,Z 609.89,A -85,B 0,C 180,E1 -29087.706,E2 -29087.706} C_VEL
LIN {X 0,Y 210.081,Z 606.338,A -85,B 0,C 180,E1 -29091.516,E2 -29091.516} C_VEL
LIN {X 0,Y 213.589,Z 601.287,A -85,B 0,C 180,E1 -29095.235,E2 -29095.235} C_VEL
LIN {X 0,Y 216.691,Z 596.354,A -85,B 0,C 180,E1 -29097.951,E2 -29097.951} C_VEL
LIN {X 0,Y 220.767,Z 589.244,A -85,B 0,C 180,E1 -29101.056,E2 -29101.056} C_VEL
LIN {X 0,Y 225.373,Z 580.491,A -85,B 0,C 180,E1 -29104.017,E2 -29104.017} C_VEL
LIN {X 0,Y 229.782,Z 571.21,A -85,B 0,C 180,E1 -29106.472,E2 -29106.472} C_VEL
LIN {X 0,Y 233.848,Z 560.924,A -85,B 0,C 180,E1 -29108.699,E2 -29108.699} C_VEL
LIN {X 0,Y 237.927,Z 549.494,A -85,B 0,C 180,E1 -29110.644,E2 -29110.644} C_VEL
LIN {X 0,Y 241.821,Z 536.78,A -85,B 0,C 180,E1 -29112.334,E2 -29112.334} C_VEL
LIN {X 0,Y 244.556,Z 524.846,A -85,B 0,C 180,E1 -29113.633,E2 -29113.633} C_VEL
LIN {X 0,Y 246.99,Z 511.131,A -85,B 0,C 180,E1 -29114.783,E2 -29114.783} C_VEL
LIN {X 0,Y 248.701,Z 497.492,A -85,B 0,C 180,E1 -29115.611,E2 -29115.611} C_VEL
LIN {X 0,Y 249.709,Z 483.229,A -85,B 0,C 180,E1 -29116.19,E2 -29116.19} C_VEL
LIN {X 0,Y 251.729,Z 444.244,A -85,B 0,C 180,E1 -29117.275,E2 -29117.275} C_VEL
LIN {X 0,Y 244.33,Z 430.028,A -85,B 0,C 180,E1 -29119.663,E2 -29119.663} C_VEL
LIN {X 0,Y 236.851,Z 417.343,A -85,B 0,C 180,E1 -29122.28,E2 -29122.28} C_VEL
LIN {X 0,Y 229.249,Z 405.827,A -85,B 0,C 180,E1 -29125.22,E2 -29125.22} C_VEL
LIN {X 0,Y 223.594,Z 397.904,A -85,B 0,C 180,E1 -29127.652,E2 -29127.652} C_VEL
LIN {X 0,Y 219.925,Z 393.142,A -85,B 0,C 180,E1 -29129.363,E2 -29129.363} C_VEL
LIN {X 0,Y 217.147,Z 389.429,A -85,B 0,C 180,E1 -29130.762,E2 -29130.762} C_VEL
LIN {X 0,Y 213.853,Z 385.662,A -85,B 0,C 180,E1 -29132.508,E2 -29132.508} C_VEL
LIN {X 0,Y 212.606,Z 383.703,A -85,B 0,C 180,E1 -29133.245,E2 -29133.245} C_VEL
LIN {X 0,Y 210.604,Z 382.001,A -85,B 0,C 180,E1 -29134.382,E2 -29134.382} C_VEL
LIN {X 0,Y 208.88,Z 385.81,A -85,B 0,C 180,E1 -29135.019,E2 -29135.019} C_VEL
LIN {X 0,Y 208.09,Z 386.72,A -85,B 0,C 180,E1 -29135.382,E2 -29135.382} C_VEL
LIN {X 0,Y 207.686,Z 386.85,A -85,B 0,C 180,E1 -29135.597,E2 -29135.597} C_VEL
LIN {X 0,Y 206.794,Z 386.162,A -85,B 0,C 180,E1 -29136.156,E2 -29136.156} C_VEL
LIN {X 0,Y 206.438,Z 384.93,A -85,B 0,C 180,E1 -29136.46,E2 -29136.46} C_VEL
LIN {X 0,Y 209.059,Z 396.133,A -85,B 0,C 180,E1 -29137.15,E2 -29137.15} C_VEL
LIN {X 0,Y 206.981,Z 473.645,A -85,B 0,C 180,E1 -29142.053,E2 -29142.053} C_VEL
LIN {X 0,Y 206.323,Z 494.514,A -85,B 0,C 180,E1 -29143.544,E2 -29143.544} C_VEL
LIN {X 0,Y 205.527,Z 510.954,A -85,B 0,C 180,E1 -29145.19,E2 -29145.19} C_VEL
LIN {X 0,Y 204.769,Z 526.134,A -85,B 0,C 180,E1 -29147.153,E2 -29147.153} C_VEL
LIN {X 0,Y 204.08,Z 539.918,A -85,B 0,C 180,E1 -29149.369,E2 -29149.369} C_VEL
LIN {X 0,Y 203.448,Z 552.477,A -85,B 0,C 180,E1 -29151.835,E2 -29151.835} C_VEL
LIN {X 0,Y 202.989,Z 564.046,A -85,B 0,C 180,E1 -29154.554,E2 -29154.554} C_VEL
LIN {X 0,Y 202.905,Z 574.744,A -85,B 0,C 180,E1 -29157.526,E2 -29157.526} C_VEL
LIN {X 0,Y 203.006,Z 583.813,A -85,B 0,C 180,E1 -29160.494,E2 -29160.494} C_VEL
LIN {X 0,Y 203.817,Z 593.859,A -85,B 0,C 180,E1 -29164.434,E2 -29164.434} C_VEL
LIN {X 0,Y 205.307,Z 601.213,A -85,B 0,C 180,E1 -29167.843,E2 -29167.843} C_VEL
LIN {X 0,Y 207.908,Z 608.104,A -85,B 0,C 180,E1 -29171.662,E2 -29171.662} C_VEL
LIN {X 0,Y 211.415,Z 613.597,A -85,B 0,C 180,E1 -29175.369,E2 -29175.369} C_VEL
LIN {X 0,Y 216.101,Z 617.77,A -85,B 0,C 180,E1 -29178.912,E2 -29178.912} C_VEL
LIN {X 0,Y 222.014,Z 620.691,A -85,B 0,C 180,E1 -29182.246,E2 -29182.246} C_VEL
LIN {X 0,Y 228.697,Z 622.378,A -85,B 0,C 180,E1 -29185.39,E2 -29185.39} C_VEL
LIN {X 0,Y 236.061,Z 622.851,A -85,B 0,C 180,E1 -29188.343,E2 -29188.343} C_VEL
LIN {X 0,Y 244.182,Z 622.113,A -85,B 0,C 180,E1 -29191.086,E2 -29191.086} C_VEL
LIN {X 0,Y 252.934,Z 620.12,A -85,B 0,C 180,E1 -29193.632,E2 -29193.632} C_VEL
LIN {X 0,Y 262.29,Z 616.865,A -85,B 0,C 180,E1 -29195.98,E2 -29195.98} C_VEL
LIN {X 0,Y 272.09,Z 612.272,A -85,B 0,C 180,E1 -29198.158,E2 -29198.158} C_VEL
LIN {X 0,Y 282.47,Z 606.153,A -85,B 0,C 180,E1 -29200.145,E2 -29200.145} C_VEL
LIN {X 0,Y 293.34,Z 598.338,A -85,B 0,C 180,E1 -29202.013,E2 -29202.013} C_VEL
LIN {X 0,Y 293.63,Z 598.235,A -85,B 0,C 180,E1 -29202.311,E2 -29202.311} C_VEL
LIN {X 0,Y 286.605,Z 604.59,A -85,B 0,C 180,E1 -29203.143,E2 -29203.143} C_VEL
LIN {X 0,Y 282.249,Z 608.188,A -85,B 0,C 180,E1 -29203.54,E2 -29203.54} C_VEL
LIN {X 0,Y 274.309,Z 613.82,A -85,B 0,C 180,E1 -29203.938,E2 -29203.938} C_VEL
LIN {X 0,Y 266.252,Z 618.902,A -85,B 0,C 180,E1 -29204.43,E2 -29204.43} C_VEL
LIN {X 0,Y 261.752,Z 621.589,A -85,B 0,C 180,E1 -29204.984,E2 -29204.984} C_VEL
LIN {X 0,Y 251.256,Z 627.634,A -85,B 0,C 180,E1 -29206.921,E2 -29206.921} C_VEL
LIN {X 0,Y 241.145,Z 632.628,A -85,B 0,C 180,E1 -29209.19,E2 -29209.19} C_VEL
LIN {X 0,Y 234.069,Z 635.679,A -85,B 0,C 180,E1 -29211.066,E2 -29211.066} C_VEL
LIN {X 0,Y 225.439,Z 638.76,A -85,B 0,C 180,E1 -29213.819,E2 -29213.819} C_VEL
LIN {X 0,Y 217.787,Z 640.833,A -85,B 0,C 180,E1 -29216.855,E2 -29216.855} C_VEL
LIN {X 0,Y 211.171,Z 641.944,A -85,B 0,C 180,E1 -29220.162,E2 -29220.162} C_VEL
LIN {X 0,Y 205.761,Z 642.142,A -85,B 0,C 180,E1 -29223.733,E2 -29223.733} C_VEL
LIN {X 0,Y 201.646,Z 641.574,A -85,B 0,C 180,E1 -29227.67,E2 -29227.67} C_VEL
LIN {X 0,Y 198.149,Z 647.113,A -85,B 0,C 180,E1 -29231.449,E2 -29231.449} C_VEL
LIN {X 0,Y 195.809,Z 651.363,A -85,B 0,C 180,E1 -29235.498,E2 -29235.498} C_VEL
LIN {X 0,Y 195.012,Z 654.26,A -85,B 0,C 180,E1 -29239.654,E2 -29239.654} C_VEL
LIN {X 0,Y 195.762,Z 655.88,A -85,B 0,C 180,E1 -29243.838,E2 -29243.838} C_VEL
LIN {X 0,Y 196.953,Z 656.359,A -85,B 0,C 180,E1 -29246.375,E2 -29246.375} C_VEL
LIN {X 0,Y 196.978,Z 664.814,A -85,B 0,C 180,E1 -29248.981,E2 -29248.981} C_VEL
LIN {X 0,Y 196.75,Z 673.005,A -85,B 0,C 180,E1 -29252.04,E2 -29252.04} C_VEL
LIN {X 0,Y 196.346,Z 679.693,A -85,B 0,C 180,E1 -29255.116,E2 -29255.116} C_VEL
LIN {X 0,Y 196.269,Z 686.964,A -85,B 0,C 180,E1 -29259.241,E2 -29259.241} C_VEL
LIN {X 0,Y 197.226,Z 692.797,A -85,B 0,C 180,E1 -29263.347,E2 -29263.347} C_VEL
LIN {X 0,Y 199.521,Z 697.424,A -85,B 0,C 180,E1 -29267.361,E2 -29267.361} C_VEL
LIN {X 0,Y 202.207,Z 700.165,A -85,B 0,C 180,E1 -29270.267,E2 -29270.267} C_VEL
LIN {X 0,Y 206.707,Z 702.88,A -85,B 0,C 180,E1 -29273.993,E2 -29273.993} C_VEL
LIN {X 0,Y 212.183,Z 704.535,A -85,B 0,C 180,E1 -29277.526,E2 -29277.526} C_VEL
LIN {X 0,Y 218.898,Z 705.142,A -85,B 0,C 180,E1 -29280.795,E2 -29280.795} C_VEL
LIN {X 0,Y 226.678,Z 704.698,A -85,B 0,C 180,E1 -29283.794,E2 -29283.794} C_VEL
LIN {X 0,Y 236.24,Z 702.969,A -85,B 0,C 180,E1 -29286.819,E2 -29286.819} C_VEL
LIN {X 0,Y 244.592,Z 700.594,A -85,B 0,C 180,E1 -29289.051,E2 -29289.051} C_VEL
LIN {X 0,Y 254.687,Z 696.818,A -85,B 0,C 180,E1 -29291.304,E2 -29291.304} C_VEL
LIN {X 0,Y 265.357,Z 691.802,A -85,B 0,C 180,E1 -29293.338,E2 -29293.338} C_VEL
LIN {X 0,Y 275.235,Z 686.277,A -85,B 0,C 180,E1 -29294.944,E2 -29294.944} C_VEL
LIN {X 0,Y 274.526,Z 686.709,A -85,B 0,C 180,E1 -29295.273,E2 -29295.273} C_VEL
LIN {X 0,Y 262.983,Z 692.971,A -85,B 0,C 180,E1 -29297.221,E2 -29297.221} C_VEL
LIN {X 0,Y 252.431,Z 697.659,A -85,B 0,C 180,E1 -29299.302,E2 -29299.302} C_VEL
LIN {X 0,Y 244.939,Z 700.336,A -85,B 0,C 180,E1 -29301.015,E2 -29301.015} C_VEL
LIN {X 0,Y 235.582,Z 702.914,A -85,B 0,C 180,E1 -29303.513,E2 -29303.513} C_VEL
LIN {X 0,Y 227.042,Z 704.392,A -85,B 0,C 180,E1 -29306.268,E2 -29306.268} C_VEL
LIN {X 0,Y 219.339,Z 704.815,A -85,B 0,C 180,E1 -29309.273,E2 -29309.273} C_VEL
LIN {X 0,Y 212.526,Z 704.177,A -85,B 0,C 180,E1 -29312.522,E2 -29312.522} C_VEL
LIN {X 0,Y 206.956,Z 702.482,A -85,B 0,C 180,E1 -29316.038,E2 -29316.038} C_VEL
LIN {X 0,Y 202.377,Z 699.733,A -85,B 0,C 180,E1 -29319.751,E2 -29319.751} C_VEL
LIN {X 0,Y 198.992,Z 695.903,A -85,B 0,C 180,E1 -29323.645,E2 -29323.645} C_VEL
LIN {X 0,Y 196.828,Z 690.914,A -85,B 0,C 180,E1 -29327.672,E2 -29327.672} C_VEL
LIN {X 0,Y 196.141,Z 684.74,A -85,B 0,C 180,E1 -29331.788,E2 -29331.788} C_VEL
LIN {X 0,Y 196.252,Z 677.016,A -85,B 0,C 180,E1 -29335.907,E2 -29335.907} C_VEL
LIN {X 0,Y 196.636,Z 669.939,A -85,B 0,C 180,E1 -29338.98,E2 -29338.98} C_VEL
LIN {X 0,Y 196.828,Z 661.254,A -85,B 0,C 180,E1 -29342.04,E2 -29342.04} C_VEL
LIN {X 0,Y 196.927,Z 651.342,A -85,B 0,C 180,E1 -29344.926,E2 -29344.926} C_VEL
LIN {X 0,Y 197.228,Z 641.061,A -85,B 0,C 180,E1 -29347.436,E2 -29347.436} C_VEL
LIN {X 0,Y 197.673,Z 628.74,A -85,B 0,C 180,E1 -29349.948,E2 -29349.948} C_VEL
LIN {X 0,Y 198.248,Z 615.059,A -85,B 0,C 180,E1 -29352.24,E2 -29352.24} C_VEL
LIN {X 0,Y 198.998,Z 599.664,A -85,B 0,C 180,E1 -29354.265,E2 -29354.265} C_VEL
LIN {X 0,Y 199.579,Z 583.908,A -85,B 0,C 180,E1 -29355.849,E2 -29355.849} C_VEL
LIN {X 0,Y 200.423,Z 556.217,A -85,B 0,C 180,E1 -29357.873,E2 -29357.873} C_VEL
LIN {X 0,Y 203.033,Z 480.98,A -85,B 0,C 180,E1 -29363.006,E2 -29363.006} C_VEL
LIN {X 0,Y 201.202,Z 453.483,A -85,B 0,C 180,E1 -29364.791,E2 -29364.791} C_VEL
LIN {X 0,Y 200.983,Z 439.651,A -85,B 0,C 180,E1 -29365.699,E2 -29365.699} C_VEL
LIN {X 0,Y 204.408,Z 412.635,A -85,B 0,C 180,E1 -29371.794,E2 -29371.794} C_VEL
LIN {X 0,Y 204.752,Z 410.313,A -85,B 0,C 180,E1 -29372.312,E2 -29372.312} C_VEL
LIN {X 0,Y 200.558,Z 390.838,A -85,B 0,C 180,E1 -29376.975,E2 -29376.975} C_VEL
LIN {X 0,Y 196.841,Z 373.511,A -85,B 0,C 180,E1 -29381.367,E2 -29381.367} C_VEL
LIN {X 0,Y 196.749,Z 373.546,A -85,B 0,C 180,E1 -29387.03,E2 -29387.03} C_VEL
LIN {X 0,Y 197.686,Z 376.286,A -85,B 0,C 180,E1 -29387.455,E2 -29387.455} C_VEL
LIN {X 0,Y 199.989,Z 378.911,A -85,B 0,C 180,E1 -29388.266,E2 -29388.266} C_VEL
LIN {X 0,Y 201.942,Z 382.04,A -85,B 0,C 180,E1 -29388.974,E2 -29388.974} C_VEL
LIN {X 0,Y 203.54,Z 384.35,A -85,B 0,C 180,E1 -29389.525,E2 -29389.525} C_VEL
LIN {X 0,Y 210.799,Z 395.424,A -85,B 0,C 180,E1 -29391.894,E2 -29391.894} C_VEL
LIN {X 0,Y 218.024,Z 407.848,A -85,B 0,C 180,E1 -29394.079,E2 -29394.079} C_VEL
LIN {X 0,Y 225.251,Z 422.101,A -85,B 0,C 180,E1 -29396.135,E2 -29396.135} C_VEL
LIN {X 0,Y 227.57,Z 427.299,A -85,B 0,C 180,E1 -29396.78,E2 -29396.78} C_VEL
LIN {X 0,Y 225.639,Z 470.756,A -85,B 0,C 180,E1 -29398.095,E2 -29398.095} C_VEL
LIN {X 0,Y 224.879,Z 490.477,A -85,B 0,C 180,E1 -29398.785,E2 -29398.785} C_VEL
LIN {X 0,Y 223.699,Z 505.012,A -85,B 0,C 180,E1 -29399.619,E2 -29399.619} C_VEL
LIN {X 0,Y 221.983,Z 518.464,A -85,B 0,C 180,E1 -29400.72,E2 -29400.72} C_VEL
LIN {X 0,Y 219.571,Z 532.03,A -85,B 0,C 180,E1 -29402.19,E2 -29402.19} C_VEL
LIN {X 0,Y 217.105,Z 544.171,A -85,B 0,C 180,E1 -29403.923,E2 -29403.923} C_VEL
LIN {X 0,Y 214.043,Z 556.462,A -85,B 0,C 180,E1 -29406.111,E2 -29406.111} C_VEL
LIN {X 0,Y 210.737,Z 567.457,A -85,B 0,C 180,E1 -29408.555,E2 -29408.555} C_VEL
LIN {X 0,Y 207.502,Z 577.324,A -85,B 0,C 180,E1 -29411.296,E2 -29411.296} C_VEL
LIN {X 0,Y 204.708,Z 585.515,A -85,B 0,C 180,E1 -29414.114,E2 -29414.114} C_VEL
LIN {X 0,Y 202.34,Z 592.355,A -85,B 0,C 180,E1 -29416.997,E2 -29416.997} C_VEL
LIN {X 0,Y 200.23,Z 598.029,A -85,B 0,C 180,E1 -29419.927,E2 -29419.927} C_VEL
LIN {X 0,Y 198.677,Z 602.679,A -85,B 0,C 180,E1 -29422.912,E2 -29422.912} C_VEL
LIN {X 0,Y 197.023,Z 607.533,A -85,B 0,C 180,E1 -29426.943,E2 -29426.943} C_VEL
LIN {X 0,Y 196.383,Z 610.195,A -85,B 0,C 180,E1 -29430,E2 -29430} C_VEL
LIN {X 0,Y 196.16,Z 612.547,A -85,B 0,C 180,E1 -29434.096,E2 -29434.096} C_VEL
LIN {X 0,Y 196.524,Z 613.609,A -85,B 0,C 180,E1 -29438.197,E2 -29438.197} C_VEL
LIN {X 0,Y 197.505,Z 613.39,A -85,B 0,C 180,E1 -29442.286,E2 -29442.286} C_VEL
LIN {X 0,Y 199.256,Z 611.867,A -85,B 0,C 180,E1 -29446.334,E2 -29446.334} C_VEL
LIN {X 0,Y 201.917,Z 608.979,A -85,B 0,C 180,E1 -29450.298,E2 -29450.298} C_VEL
LIN {X 0,Y 205.244,Z 604.662,A -85,B 0,C 180,E1 -29454.176,E2 -29454.176} C_VEL
LIN {X 0,Y 208.223,Z 600.348,A -85,B 0,C 180,E1 -29457.009,E2 -29457.009} C_VEL
LIN {X 0,Y 211.607,Z 595.074,A -85,B 0,C 180,E1 -29459.77,E2 -29459.77} C_VEL
LIN {X 0,Y 216.003,Z 587.484,A -85,B 0,C 180,E1 -29462.899,E2 -29462.899} C_VEL
LIN {X 0,Y 220.222,Z 579.52,A -85,B 0,C 180,E1 -29465.484,E2 -29465.484} C_VEL
LIN {X 0,Y 224.868,Z 569.88,A -85,B 0,C 180,E1 -29467.967,E2 -29467.967} C_VEL
LIN {X 0,Y 228.892,Z 559.847,A -85,B 0,C 180,E1 -29470.089,E2 -29470.089} C_VEL
LIN {X 0,Y 233.04,Z 548.489,A -85,B 0,C 180,E1 -29471.972,E2 -29471.972} C_VEL
LIN {X 0,Y 236.6,Z 536.949,A -85,B 0,C 180,E1 -29473.497,E2 -29473.497} C_VEL
LIN {X 0,Y 239.711,Z 523.63,A -85,B 0,C 180,E1 -29474.93,E2 -29474.93} C_VEL
LIN {X 0,Y 242.062,Z 510.366,A -85,B 0,C 180,E1 -29476.014,E2 -29476.014} C_VEL
LIN {X 0,Y 243.781,Z 496.518,A -85,B 0,C 180,E1 -29476.824,E2 -29476.824} C_VEL
LIN {X 0,Y 244.732,Z 481.236,A -85,B 0,C 180,E1 -29477.419,E2 -29477.419} C_VEL
LIN {X 0,Y 246.614,Z 446.859,A -85,B 0,C 180,E1 -29478.382,E2 -29478.382} C_VEL
LIN {X 0,Y 238.924,Z 432.072,A -85,B 0,C 180,E1 -29481.017,E2 -29481.017} C_VEL
LIN {X 0,Y 231.42,Z 419.456,A -85,B 0,C 180,E1 -29483.827,E2 -29483.827} C_VEL
LIN {X 0,Y 223.846,Z 408.013,A -85,B 0,C 180,E1 -29486.998,E2 -29486.998} C_VEL
LIN {X 0,Y 217.635,Z 399.497,A -85,B 0,C 180,E1 -29489.93,E2 -29489.93} C_VEL
LIN {X 0,Y 214.604,Z 395.461,A -85,B 0,C 180,E1 -29491.512,E2 -29491.512} C_VEL
LIN {X 0,Y 211.299,Z 391.498,A -85,B 0,C 180,E1 -29493.352,E2 -29493.352} C_VEL
LIN {X 0,Y 211.111,Z 391.171,A -85,B 0,C 180,E1 -29493.47,E2 -29493.47} C_VEL
LIN {X 0,Y 210.279,Z 391.348,A -85,B 0,C 180,E1 -29493.879,E2 -29493.879} C_VEL
LIN {X 0,Y 208.329,Z 393.432,A -85,B 0,C 180,E1 -29494.749,E2 -29494.749} C_VEL
LIN {X 0,Y 207.839,Z 393.675,A -85,B 0,C 180,E1 -29494.996,E2 -29494.996} C_VEL
LIN {X 0,Y 204.433,Z 404.508,A -85,B 0,C 180,E1 -29496.074,E2 -29496.074} C_VEL
LIN {X 0,Y 202.752,Z 408.22,A -85,B 0,C 180,E1 -29496.77,E2 -29496.77} C_VEL
LIN {X 0,Y 201.988,Z 408.762,A -85,B 0,C 180,E1 -29497.191,E2 -29497.191} C_VEL
LIN {X 0,Y 201.695,Z 407.522,A -85,B 0,C 180,E1 -29497.477,E2 -29497.477} C_VEL
LIN {X 0,Y 201.679,Z 404.529,A -85,B 0,C 180,E1 -29497.741,E2 -29497.741} C_VEL
LIN {X 0,Y 199.962,Z 472.957,A -85,B 0,C 180,E1 -29502.283,E2 -29502.283} C_VEL
LIN {X 0,Y 199.279,Z 494.548,A -85,B 0,C 180,E1 -29503.865,E2 -29503.865} C_VEL
LIN {X 0,Y 198.552,Z 510.057,A -85,B 0,C 180,E1 -29505.442,E2 -29505.442} C_VEL
LIN {X 0,Y 197.807,Z 525.513,A -85,B 0,C 180,E1 -29507.473,E2 -29507.473} C_VEL
LIN {X 0,Y 197.123,Z 539.323,A -85,B 0,C 180,E1 -29509.766,E2 -29509.766} C_VEL
LIN {X 0,Y 196.52,Z 552.041,A -85,B 0,C 180,E1 -29512.318,E2 -29512.318} C_VEL
LIN {X 0,Y 196.082,Z 564.816,A -85,B 0,C 180,E1 -29515.389,E2 -29515.389} C_VEL
LIN {X 0,Y 196.052,Z 575.446,A -85,B 0,C 180,E1 -29518.464,E2 -29518.464} C_VEL
LIN {X 0,Y 196.295,Z 585.778,A -85,B 0,C 180,E1 -29522.044,E2 -29522.044} C_VEL
LIN {X 0,Y 197.379,Z 595.697,A -85,B 0,C 180,E1 -29526.111,E2 -29526.111} C_VEL
LIN {X 0,Y 199.594,Z 603.764,A -85,B 0,C 180,E1 -29530.105,E2 -29530.105} C_VEL
LIN {X 0,Y 202.681,Z 610.354,A -85,B 0,C 180,E1 -29533.999,E2 -29533.999} C_VEL
LIN {X 0,Y 206.836,Z 615.553,A -85,B 0,C 180,E1 -29537.745,E2 -29537.745} C_VEL
LIN {X 0,Y 212.32,Z 619.531,A -85,B 0,C 180,E1 -29541.277,E2 -29541.277} C_VEL
LIN {X 0,Y 218.807,Z 622.236,A -85,B 0,C 180,E1 -29544.592,E2 -29544.592} C_VEL
LIN {X 0,Y 226.037,Z 623.748,A -85,B 0,C 180,E1 -29547.698,E2 -29547.698} C_VEL
LIN {X 0,Y 233.959,Z 624.066,A -85,B 0,C 180,E1 -29550.594,E2 -29550.594} C_VEL
LIN {X 0,Y 243.764,Z 622.972,A -85,B 0,C 180,E1 -29553.56,E2 -29553.56} C_VEL
LIN {X 0,Y 252.007,Z 621.02,A -85,B 0,C 180,E1 -29555.71,E2 -29555.71} C_VEL
LIN {X 0,Y 261.836,Z 617.626,A -85,B 0,C 180,E1 -29557.972,E2 -29557.972} C_VEL
LIN {X 0,Y 272.188,Z 612.85,A -85,B 0,C 180,E1 -29560.041,E2 -29560.041} C_VEL
LIN {X 0,Y 283.023,Z 606.593,A -85,B 0,C 180,E1 -29561.929,E2 -29561.929} C_VEL
LIN {X 0,Y 270.713,Z 615.736,A -85,B 0,C 180,E1 -29563.574,E2 -29563.574} C_VEL
LIN {X 0,Y 261.752,Z 621.589,A -85,B 0,C 180,E1 -29564.984,E2 -29564.984} C_VEL
LIN {X 0,Y 257.157,Z 624.183,A -85,B 0,C 180,E1 -29565.594,E2 -29565.594} C_VEL
LIN {X 0,Y 248.663,Z 628.098,A -85,B 0,C 180,E1 -29566.363,E2 -29566.363} C_VEL
LIN {X 0,Y 240.231,Z 631.357,A -85,B 0,C 180,E1 -29567.261,E2 -29567.261} C_VEL
LIN {X 0,Y 235.79,Z 633.017,A -85,B 0,C 180,E1 -29568.081,E2 -29568.081} C_VEL
LIN {X 0,Y 228.589,Z 635.672,A -85,B 0,C 180,E1 -29569.947,E2 -29569.947} C_VEL
LIN {X 0,Y 219.778,Z 638.319,A -85,B 0,C 180,E1 -29572.732,E2 -29572.732} C_VEL
LIN {X 0,Y 211.908,Z 640.005,A -85,B 0,C 180,E1 -29575.811,E2 -29575.811} C_VEL
LIN {X 0,Y 205.122,Z 640.78,A -85,B 0,C 180,E1 -29579.188,E2 -29579.188} C_VEL
LIN {X 0,Y 199.543,Z 640.601,A -85,B 0,C 180,E1 -29582.849,E2 -29582.849} C_VEL
LIN {X 0,Y 195.851,Z 639.913,A -85,B 0,C 180,E1 -29586.275,E2 -29586.275} C_VEL
LIN {X 0,Y 192.226,Z 645.156,A -85,B 0,C 180,E1 -29589.747,E2 -29589.747} C_VEL
LIN {X 0,Y 189.997,Z 648.731,A -85,B 0,C 180,E1 -29592.846,E2 -29592.846} C_VEL
LIN {X 0,Y 188.241,Z 652.255,A -85,B 0,C 180,E1 -29597.099,E2 -29597.099} C_VEL
LIN {X 0,Y 188.089,Z 654.47,A -85,B 0,C 180,E1 -29601.433,E2 -29601.433} C_VEL
LIN {X 0,Y 189.58,Z 655.433,A -85,B 0,C 180,E1 -29606.004,E2 -29606.004} C_VEL
LIN {X 0,Y 190.27,Z 655.556,A -85,B 0,C 180,E1 -29607.111,E2 -29607.111} C_VEL
LIN {X 0,Y 190.316,Z 663.077,A -85,B 0,C 180,E1 -29609.472,E2 -29609.472} C_VEL
LIN {X 0,Y 190.077,Z 671.431,A -85,B 0,C 180,E1 -29612.662,E2 -29612.662} C_VEL
LIN {X 0,Y 189.631,Z 679.188,A -85,B 0,C 180,E1 -29616.362,E2 -29616.362} C_VEL
LIN {X 0,Y 189.778,Z 686.44,A -85,B 0,C 180,E1 -29620.634,E2 -29620.634} C_VEL
LIN {X 0,Y 191.066,Z 692.29,A -85,B 0,C 180,E1 -29624.869,E2 -29624.869} C_VEL
LIN {X 0,Y 193.706,Z 696.958,A -85,B 0,C 180,E1 -29628.992,E2 -29628.992} C_VEL
LIN {X 0,Y 198.361,Z 700.911,A -85,B 0,C 180,E1 -29633.351,E2 -29633.351} C_VEL
LIN {X 0,Y 203.017,Z 703.097,A -85,B 0,C 180,E1 -29636.649,E2 -29636.649} C_VEL
LIN {X 0,Y 209.246,Z 704.619,A -85,B 0,C 180,E1 -29640.14,E2 -29640.14} C_VEL
LIN {X 0,Y 216.713,Z 705.138,A -85,B 0,C 180,E1 -29643.33,E2 -29643.33} C_VEL
LIN {X 0,Y 225.136,Z 704.579,A -85,B 0,C 180,E1 -29646.237,E2 -29646.237} C_VEL
LIN {X 0,Y 234.303,Z 702.974,A -85,B 0,C 180,E1 -29648.887,E2 -29648.887} C_VEL
LIN {X 0,Y 244.223,Z 700.286,A -85,B 0,C 180,E1 -29651.273,E2 -29651.273} C_VEL
LIN {X 0,Y 254.852,Z 696.429,A -85,B 0,C 180,E1 -29653.401,E2 -29653.401} C_VEL
LIN {X 0,Y 263.168,Z 692.766,A -85,B 0,C 180,E1 -29654.851,E2 -29654.851} C_VEL
LIN {X 0,Y 262.432,Z 693.095,A -85,B 0,C 180,E1 -29655.403,E2 -29655.403} C_VEL
LIN {X 0,Y 252.467,Z 697.362,A -85,B 0,C 180,E1 -29657.178,E2 -29657.178} C_VEL
LIN {X 0,Y 244.579,Z 700.087,A -85,B 0,C 180,E1 -29658.8,E2 -29658.8} C_VEL
LIN {X 0,Y 234.644,Z 702.756,A -85,B 0,C 180,E1 -29661.18,E2 -29661.18} C_VEL
LIN {X 0,Y 225.465,Z 704.337,A -85,B 0,C 180,E1 -29663.824,E2 -29663.824} C_VEL
LIN {X 0,Y 217.111,Z 704.862,A -85,B 0,C 180,E1 -29666.739,E2 -29666.739} C_VEL
LIN {X 0,Y 209.625,Z 704.314,A -85,B 0,C 180,E1 -29669.92,E2 -29669.92} C_VEL
LIN {X 0,Y 203.276,Z 702.758,A -85,B 0,C 180,E1 -29673.388,E2 -29673.388} C_VEL
LIN {X 0,Y 198.073,Z 700.201,A -85,B 0,C 180,E1 -29677.109,E2 -29677.109} C_VEL
LIN {X 0,Y 193.859,Z 696.557,A -85,B 0,C 180,E1 -29681.024,E2 -29681.024} C_VEL
LIN {X 0,Y 191.128,Z 691.852,A -85,B 0,C 180,E1 -29685.136,E2 -29685.136} C_VEL
LIN {X 0,Y 189.656,Z 685.936,A -85,B 0,C 180,E1 -29689.359,E2 -29689.359} C_VEL
LIN {X 0,Y 189.416,Z 680.628,A -85,B 0,C 180,E1 -29692.564,E2 -29692.564} C_VEL
LIN {X 0,Y 189.771,Z 672.096,A -85,B 0,C 180,E1 -29696.827,E2 -29696.827} C_VEL
LIN {X 0,Y 190.082,Z 664.093,A -85,B 0,C 180,E1 -29700.001,E2 -29700.001} C_VEL
LIN {X 0,Y 190.189,Z 656.091,A -85,B 0,C 180,E1 -29702.639,E2 -29702.639} C_VEL
LIN {X 0,Y 190.394,Z 643.464,A -85,B 0,C 180,E1 -29706.072,E2 -29706.072} C_VEL
LIN {X 0,Y 190.819,Z 630.256,A -85,B 0,C 180,E1 -29708.976,E2 -29708.976} C_VEL
LIN {X 0,Y 191.343,Z 615.252,A -85,B 0,C 180,E1 -29711.616,E2 -29711.616} C_VEL
LIN {X 0,Y 192.044,Z 600.084,A -85,B 0,C 180,E1 -29713.715,E2 -29713.715} C_VEL
LIN {X 0,Y 192.609,Z 584.735,A -85,B 0,C 180,E1 -29715.355,E2 -29715.355} C_VEL
LIN {X 0,Y 193.332,Z 559.216,A -85,B 0,C 180,E1 -29717.324,E2 -29717.324} C_VEL
LIN {X 0,Y 195.926,Z 481.129,A -85,B 0,C 180,E1 -29722.914,E2 -29722.914} C_VEL
LIN {X 0,Y 194.015,Z 451.408,A -85,B 0,C 180,E1 -29724.923,E2 -29724.923} C_VEL
LIN {X 0,Y 193.91,Z 439.523,A -85,B 0,C 180,E1 -29725.76,E2 -29725.76} C_VEL
LIN {X 0,Y 197.326,Z 413.041,A -85,B 0,C 180,E1 -29731.914,E2 -29731.914} C_VEL
LIN {X 0,Y 197.616,Z 410.88,A -85,B 0,C 180,E1 -29732.411,E2 -29732.411} C_VEL
LIN {X 0,Y 193.672,Z 392.516,A -85,B 0,C 180,E1 -29736.92,E2 -29736.92} C_VEL
LIN {X 0,Y 189.786,Z 374.391,A -85,B 0,C 180,E1 -29741.632,E2 -29741.632} C_VEL
LIN {X 0,Y 189.676,Z 374.406,A -85,B 0,C 180,E1 -29744.781,E2 -29744.781} C_VEL
LIN {X 0,Y 190.636,Z 377.185,A -85,B 0,C 180,E1 -29745.266,E2 -29745.266} C_VEL
LIN {X 0,Y 193.128,Z 379.972,A -85,B 0,C 180,E1 -29746.235,E2 -29746.235} C_VEL
LIN {X 0,Y 195.338,Z 383.33,A -85,B 0,C 180,E1 -29747.107,E2 -29747.107} C_VEL
LIN {X 0,Y 196.727,Z 385.287,A -85,B 0,C 180,E1 -29747.63,E2 -29747.63} C_VEL
LIN {X 0,Y 199.897,Z 389.971,A -85,B 0,C 180,E1 -29748.79,E2 -29748.79} C_VEL
LIN {X 0,Y 206.554,Z 400.248,A -85,B 0,C 180,E1 -29751.064,E2 -29751.064} C_VEL
LIN {X 0,Y 213.889,Z 413.082,A -85,B 0,C 180,E1 -29753.388,E2 -29753.388} C_VEL
LIN {X 0,Y 220.722,Z 426.997,A -85,B 0,C 180,E1 -29755.432,E2 -29755.432} C_VEL
LIN {X 0,Y 221.836,Z 429.413,A -85,B 0,C 180,E1 -29755.753,E2 -29755.753} C_VEL
LIN {X 0,Y 219.876,Z 471.344,A -85,B 0,C 180,E1 -29757.045,E2 -29757.045} C_VEL
LIN {X 0,Y 219.06,Z 491.371,A -85,B 0,C 180,E1 -29757.763,E2 -29757.763} C_VEL
LIN {X 0,Y 217.869,Z 505.362,A -85,B 0,C 180,E1 -29758.575,E2 -29758.575} C_VEL
LIN {X 0,Y 216.085,Z 518.965,A -85,B 0,C 180,E1 -29759.705,E2 -29759.705} C_VEL
LIN {X 0,Y 213.752,Z 531.721,A -85,B 0,C 180,E1 -29761.096,E2 -29761.096} C_VEL
LIN {X 0,Y 211.131,Z 544.076,A -85,B 0,C 180,E1 -29762.86,E2 -29762.86} C_VEL
LIN {X 0,Y 208.293,Z 555.362,A -85,B 0,C 180,E1 -29764.878,E2 -29764.878} C_VEL
LIN {X 0,Y 204.818,Z 566.725,A -85,B 0,C 180,E1 -29767.373,E2 -29767.373} C_VEL
LIN {X 0,Y 201.369,Z 576.99,A -85,B 0,C 180,E1 -29770.209,E2 -29770.209} C_VEL
LIN {X 0,Y 198.41,Z 585.285,A -85,B 0,C 180,E1 -29773.068,E2 -29773.068} C_VEL
LIN {X 0,Y 195.486,Z 593.313,A -85,B 0,C 180,E1 -29776.532,E2 -29776.532} C_VEL
LIN {X 0,Y 193.309,Z 598.965,A -85,B 0,C 180,E1 -29779.562,E2 -29779.562} C_VEL
LIN {X 0,Y 191.69,Z 603.58,A -85,B 0,C 180,E1 -29782.653,E2 -29782.653} C_VEL
LIN {X 0,Y 189.976,Z 608.401,A -85,B 0,C 180,E1 -29786.83,E2 -29786.83} C_VEL
LIN {X 0,Y 189.191,Z 612.046,A -85,B 0,C 180,E1 -29791.539,E2 -29791.539} C_VEL
LIN {X 0,Y 189.115,Z 613.353,A -85,B 0,C 180,E1 -29794.248,E2 -29794.248} C_VEL
LIN {X 0,Y 189.506,Z 614.387,A -85,B 0,C 180,E1 -29798.503,E2 -29798.503} C_VEL
LIN {X 0,Y 190.577,Z 614.139,A -85,B 0,C 180,E1 -29802.74,E2 -29802.74} C_VEL
LIN {X 0,Y 192.47,Z 612.583,A -85,B 0,C 180,E1 -29806.927,E2 -29806.927} C_VEL
LIN {X 0,Y 195.63,Z 609.315,A -85,B 0,C 180,E1 -29811.42,E2 -29811.42} C_VEL
LIN {X 0,Y 198.789,Z 605.315,A -85,B 0,C 180,E1 -29815.014,E2 -29815.014} C_VEL
LIN {X 0,Y 201.907,Z 600.968,A -85,B 0,C 180,E1 -29817.927,E2 -29817.927} C_VEL
LIN {X 0,Y 205.478,Z 595.654,A -85,B 0,C 180,E1 -29820.753,E2 -29820.753} C_VEL
LIN {X 0,Y 210.069,Z 588.022,A -85,B 0,C 180,E1 -29823.952,E2 -29823.952} C_VEL
LIN {X 0,Y 214.479,Z 580.01,A -85,B 0,C 180,E1 -29826.585,E2 -29826.585} C_VEL
LIN {X 0,Y 219.292,Z 570.315,A -85,B 0,C 180,E1 -29829.113,E2 -29829.113} C_VEL
LIN {X 0,Y 223.339,Z 560.582,A -85,B 0,C 180,E1 -29831.195,E2 -29831.195} C_VEL
LIN {X 0,Y 227.794,Z 548.771,A -85,B 0,C 180,E1 -29833.171,E2 -29833.171} C_VEL
LIN {X 0,Y 231.479,Z 537.119,A -85,B 0,C 180,E1 -29834.712,E2 -29834.712} C_VEL
LIN {X 0,Y 234.653,Z 523.902,A -85,B 0,C 180,E1 -29836.135,E2 -29836.135} C_VEL
LIN {X 0,Y 237.189,Z 509.716,A -85,B 0,C 180,E1 -29837.278,E2 -29837.278} C_VEL
LIN {X 0,Y 238.9,Z 495.845,A -85,B 0,C 180,E1 -29838.066,E2 -29838.066} C_VEL
LIN {X 0,Y 239.924,Z 479.246,A -85,B 0,C 180,E1 -29838.683,E2 -29838.683} C_VEL
LIN {X 0,Y 241.617,Z 449.597,A -85,B 0,C 180,E1 -29839.524,E2 -29839.524} C_VEL
LIN {X 0,Y 234.424,Z 435.665,A -85,B 0,C 180,E1 -29842.134,E2 -29842.134} C_VEL
LIN {X 0,Y 227.552,Z 424.055,A -85,B 0,C 180,E1 -29844.851,E2 -29844.851} C_VEL
LIN {X 0,Y 220.692,Z 413.443,A -85,B 0,C 180,E1 -29847.878,E2 -29847.878} C_VEL
LIN {X 0,Y 214.72,Z 405.158,A -85,B 0,C 180,E1 -29850.837,E2 -29850.837} C_VEL
LIN {X 0,Y 211.256,Z 400.626,A -85,B 0,C 180,E1 -29852.743,E2 -29852.743} C_VEL
LIN {X 0,Y 209.838,Z 399.154,A -85,B 0,C 180,E1 -29853.549,E2 -29853.549} C_VEL
LIN {X 0,Y 206.344,Z 409.169,A -85,B 0,C 180,E1 -29854.648,E2 -29854.648} C_VEL
LIN {X 0,Y 204.34,Z 413.284,A -85,B 0,C 180,E1 -29855.441,E2 -29855.441} C_VEL
LIN {X 0,Y 202.858,Z 415.123,A -85,B 0,C 180,E1 -29856.148,E2 -29856.148} C_VEL
LIN {X 0,Y 202.385,Z 415.445,A -85,B 0,C 180,E1 -29856.402,E2 -29856.402} C_VEL
LIN {X 0,Y 198.509,Z 430.832,A -85,B 0,C 180,E1 -29857.503,E2 -29857.503} C_VEL
LIN {X 0,Y 195.886,Z 439.489,A -85,B 0,C 180,E1 -29858.461,E2 -29858.461} C_VEL
LIN {X 0,Y 194.343,Z 443.142,A -85,B 0,C 180,E1 -29859.19,E2 -29859.19} C_VEL
LIN {X 0,Y 193.607,Z 443.543,A -85,B 0,C 180,E1 -29859.679,E2 -29859.679} C_VEL
LIN {X 0,Y 193.364,Z 442.19,A -85,B 0,C 180,E1 -29859.988,E2 -29859.988} C_VEL
LIN {X 0,Y 193.421,Z 439.58,A -85,B 0,C 180,E1 -29860.202,E2 -29860.202} C_VEL
LIN {X 0,Y 192.665,Z 483.015,A -85,B 0,C 180,E1 -29863.295,E2 -29863.295} C_VEL
LIN {X 0,Y 192.056,Z 499.077,A -85,B 0,C 180,E1 -29864.667,E2 -29864.667} C_VEL
LIN {X 0,Y 191.36,Z 514.136,A -85,B 0,C 180,E1 -29866.37,E2 -29866.37} C_VEL
LIN {X 0,Y 190.651,Z 529.549,A -85,B 0,C 180,E1 -29868.61,E2 -29868.61} C_VEL
LIN {X 0,Y 190.01,Z 542.818,A -85,B 0,C 180,E1 -29870.986,E2 -29870.986} C_VEL
LIN {X 0,Y 189.427,Z 556.177,A -85,B 0,C 180,E1 -29873.897,E2 -29873.897} C_VEL
LIN {X 0,Y 189.169,Z 569.102,A -85,B 0,C 180,E1 -29877.347,E2 -29877.347} C_VEL
LIN {X 0,Y 189.272,Z 579.148,A -85,B 0,C 180,E1 -29880.53,E2 -29880.53} C_VEL
LIN {X 0,Y 189.816,Z 589.051,A -85,B 0,C 180,E1 -29884.232,E2 -29884.232} C_VEL
LIN {X 0,Y 191.467,Z 598.414,A -85,B 0,C 180,E1 -29888.414,E2 -29888.414} C_VEL
LIN {X 0,Y 194.13,Z 606.19,A -85,B 0,C 180,E1 -29892.502,E2 -29892.502} C_VEL
LIN {X 0,Y 197.82,Z 612.476,A -85,B 0,C 180,E1 -29896.455,E2 -29896.455} C_VEL
LIN {X 0,Y 202.745,Z 617.497,A -85,B 0,C 180,E1 -29900.211,E2 -29900.211} C_VEL
LIN {X 0,Y 208.948,Z 621.249,A -85,B 0,C 180,E1 -29903.72,E2 -29903.72} C_VEL
LIN {X 0,Y 216.002,Z 623.786,A -85,B 0,C 180,E1 -29906.999,E2 -29906.999} C_VEL
LIN {X 0,Y 223.815,Z 625.13,A -85,B 0,C 180,E1 -29910.048,E2 -29910.048} C_VEL
LIN {X 0,Y 232.382,Z 625.278,A -85,B 0,C 180,E1 -29912.857,E2 -29912.857} C_VEL
LIN {X 0,Y 241.631,Z 624.232,A -85,B 0,C 180,E1 -29915.433,E2 -29915.433} C_VEL
LIN {X 0,Y 251.482,Z 621.967,A -85,B 0,C 180,E1 -29917.789,E2 -29917.789} C_VEL
LIN {X 0,Y 261.808,Z 618.424,A -85,B 0,C 180,E1 -29919.948,E2 -29919.948} C_VEL
LIN {X 0,Y 269.075,Z 615.254,A -85,B 0,C 180,E1 -29921.289,E2 -29921.289} C_VEL
LIN {X 0,Y 270.347,Z 614.84,A -85,B 0,C 180,E1 -29921.859,E2 -29921.859} C_VEL
LIN {X 0,Y 260.054,Z 621.199,A -85,B 0,C 180,E1 -29923.344,E2 -29923.344} C_VEL
LIN {X 0,Y 248.811,Z 627.22,A -85,B 0,C 180,E1 -29925.267,E2 -29925.267} C_VEL
LIN {X 0,Y 238.333,Z 632.013,A -85,B 0,C 180,E1 -29927.471,E2 -29927.471} C_VEL
LIN {X 0,Y 235.79,Z 633.017,A -85,B 0,C 180,E1 -29928.081,E2 -29928.081} C_VEL
LIN {X 0,Y 231.361,Z 634.544,A -85,B 0,C 180,E1 -29928.971,E2 -29928.971} C_VEL
LIN {X 0,Y 223.02,Z 636.497,A -85,B 0,C 180,E1 -29930.235,E2 -29930.235} C_VEL
LIN {X 0,Y 214.889,Z 637.79,A -85,B 0,C 180,E1 -29931.652,E2 -29931.652} C_VEL
LIN {X 0,Y 210.852,Z 638.343,A -85,B 0,C 180,E1 -29932.785,E2 -29932.785} C_VEL
LIN {X 0,Y 202.561,Z 639.375,A -85,B 0,C 180,E1 -29936.408,E2 -29936.408} C_VEL
LIN {X 0,Y 196.121,Z 639.278,A -85,B 0,C 180,E1 -29939.999,E2 -29939.999} C_VEL
LIN {X 0,Y 190.183,Z 638.247,A -85,B 0,C 180,E1 -29944.795,E2 -29944.795} C_VEL
LIN {X 0,Y 186.523,Z 643.125,A -85,B 0,C 180,E1 -29947.943,E2 -29947.943} C_VEL
LIN {X 0,Y 183.209,Z 648.046,A -85,B 0,C 180,E1 -29952.19,E2 -29952.19} C_VEL
LIN {X 0,Y 181.266,Z 651.53,A -85,B 0,C 180,E1 -29956.594,E2 -29956.594} C_VEL
LIN {X 0,Y 180.987,Z 653.71,A -85,B 0,C 180,E1 -29961.094,E2 -29961.094} C_VEL
LIN {X 0,Y 182.273,Z 654.638,A -85,B 0,C 180,E1 -29965.592,E2 -29965.592} C_VEL
LIN {X 0,Y 183.659,Z 654.824,A -85,B 0,C 180,E1 -29967.951,E2 -29967.951} C_VEL
LIN {X 0,Y 183.649,Z 662.701,A -85,B 0,C 180,E1 -29970.546,E2 -29970.546} C_VEL
LIN {X 0,Y 183.425,Z 670.271,A -85,B 0,C 180,E1 -29973.569,E2 -29973.569} C_VEL
LIN {X 0,Y 183.004,Z 677.584,A -85,B 0,C 180,E1 -29977.145,E2 -29977.145} C_VEL
LIN {X 0,Y 183.179,Z 684.173,A -85,B 0,C 180,E1 -29981.022,E2 -29981.022} C_VEL
LIN {X 0,Y 184.47,Z 690.365,A -85,B 0,C 180,E1 -29985.414,E2 -29985.414} C_VEL
LIN {X 0,Y 187.173,Z 695.392,A -85,B 0,C 180,E1 -29989.682,E2 -29989.682} C_VEL
LIN {X 0,Y 191.994,Z 699.752,A -85,B 0,C 180,E1 -29994.209,E2 -29994.209} C_VEL
LIN {X 0,Y 196.759,Z 702.219,A -85,B 0,C 180,E1 -29997.567,E2 -29997.567} C_VEL
LIN {X 0,Y 203.174,Z 704.094,A -85,B 0,C 180,E1 -30001.139,E2 -30001.139} C_VEL
LIN {X 0,Y 210.834,Z 705.01,A -85,B 0,C 180,E1 -30004.387,E2 -30004.387} C_VEL
LIN {X 0,Y 219.472,Z 704.917,A -85,B 0,C 180,E1 -30007.328,E2 -30007.328} C_VEL
LIN {X 0,Y 228.841,Z 703.764,A -85,B 0,C 180,E1 -30009.999,E2 -30009.999} C_VEL
LIN {X 0,Y 238.99,Z 701.546,A -85,B 0,C 180,E1 -30012.384,E2 -30012.384} C_VEL
LIN {X 0,Y 252.008,Z 697.449,A -85,B 0,C 180,E1 -30014.892,E2 -30014.892} C_VEL
LIN {X 0,Y 251.451,Z 697.638,A -85,B 0,C 180,E1 -30015.338,E2 -30015.338} C_VEL
LIN {X 0,Y 239.331,Z 701.397,A -85,B 0,C 180,E1 -30017.691,E2 -30017.691} C_VEL
LIN {X 0,Y 229.178,Z 703.594,A -85,B 0,C 180,E1 -30020.072,E2 -30020.072} C_VEL
LIN {X 0,Y 219.786,Z 704.71,A -85,B 0,C 180,E1 -30022.734,E2 -30022.734} C_VEL
LIN {X 0,Y 211.228,Z 704.777,A -85,B 0,C 180,E1 -30025.686,E2 -30025.686} C_VEL
LIN {X 0,Y 203.542,Z 703.839,A -85,B 0,C 180,E1 -30028.923,E2 -30028.923} C_VEL
LIN {X 0,Y 197.017,Z 701.927,A -85,B 0,C 180,E1 -30032.473,E2 -30032.473} C_VEL
LIN {X 0,Y 191.653,Z 699.029,A -85,B 0,C 180,E1 -30036.296,E2 -30036.296} C_VEL
LIN {X 0,Y 187.317,Z 695.027,A -85,B 0,C 180,E1 -30040.334,E2 -30040.334} C_VEL
LIN {X 0,Y 184.523,Z 689.96,A -85,B 0,C 180,E1 -30044.591,E2 -30044.591} C_VEL
LIN {X 0,Y 183.051,Z 683.704,A -85,B 0,C 180,E1 -30048.97,E2 -30048.97} C_VEL
LIN {X 0,Y 182.817,Z 676.066,A -85,B 0,C 180,E1 -30053.4,E2 -30053.4} C_VEL
LIN {X 0,Y 183.24,Z 669.2,A -85,B 0,C 180,E1 -30056.689,E2 -30056.689} C_VEL
LIN {X 0,Y 183.464,Z 662.104,A -85,B 0,C 180,E1 -30059.519,E2 -30059.519} C_VEL
LIN {X 0,Y 183.526,Z 652.537,A -85,B 0,C 180,E1 -30062.648,E2 -30062.648} C_VEL
LIN {X 0,Y 183.677,Z 641.019,A -85,B 0,C 180,E1 -30065.763,E2 -30065.763} C_VEL
LIN {X 0,Y 184.069,Z 627.455,A -85,B 0,C 180,E1 -30068.756,E2 -30068.756} C_VEL
LIN {X 0,Y 184.533,Z 613.593,A -85,B 0,C 180,E1 -30071.218,E2 -30071.218} C_VEL
LIN {X 0,Y 185.213,Z 598.242,A -85,B 0,C 180,E1 -30073.394,E2 -30073.394} C_VEL
LIN {X 0,Y 185.733,Z 582.166,A -85,B 0,C 180,E1 -30075.097,E2 -30075.097} C_VEL
LIN {X 0,Y 186.658,Z 546.655,A -85,B 0,C 180,E1 -30077.894,E2 -30077.894} C_VEL
LIN {X 0,Y 188.855,Z 481.317,A -85,B 0,C 180,E1 -30082.776,E2 -30082.776} C_VEL
LIN {X 0,Y 186.933,Z 451.401,A -85,B 0,C 180,E1 -30084.878,E2 -30084.878} C_VEL
LIN {X 0,Y 186.812,Z 439.66,A -85,B 0,C 180,E1 -30085.721,E2 -30085.721} C_VEL
LIN {X 0,Y 190.42,Z 411.812,A -85,B 0,C 180,E1 -30092.404,E2 -30092.404} C_VEL
LIN {X 0,Y 189.22,Z 405.404,A -85,B 0,C 180,E1 -30093.992,E2 -30093.992} C_VEL
LIN {X 0,Y 185.202,Z 386.921,A -85,B 0,C 180,E1 -30098.735,E2 -30098.735} C_VEL
LIN {X 0,Y 182.735,Z 375.27,A -85,B 0,C 180,E1 -30101.915,E2 -30101.915} C_VEL
LIN {X 0,Y 182.747,Z 375.376,A -85,B 0,C 180,E1 -30102.311,E2 -30102.311} C_VEL
LIN {X 0,Y 183.726,Z 378.166,A -85,B 0,C 180,E1 -30102.857,E2 -30102.857} C_VEL
LIN {X 0,Y 185.746,Z 380.278,A -85,B 0,C 180,E1 -30103.733,E2 -30103.733} C_VEL
LIN {X 0,Y 188.461,Z 384.301,A -85,B 0,C 180,E1 -30104.925,E2 -30104.925} C_VEL
LIN {X 0,Y 189.837,Z 386.053,A -85,B 0,C 180,E1 -30105.489,E2 -30105.489} C_VEL
LIN {X 0,Y 195.459,Z 394.191,A -85,B 0,C 180,E1 -30107.707,E2 -30107.707} C_VEL
LIN {X 0,Y 202.577,Z 405.422,A -85,B 0,C 180,E1 -30110.275,E2 -30110.275} C_VEL
LIN {X 0,Y 209.944,Z 418.707,A -85,B 0,C 180,E1 -30112.725,E2 -30112.725} C_VEL
LIN {X 0,Y 216.118,Z 431.645,A -85,B 0,C 180,E1 -30114.664,E2 -30114.664} C_VEL
LIN {X 0,Y 213.959,Z 477.335,A -85,B 0,C 180,E1 -30116.114,E2 -30116.114} C_VEL
LIN {X 0,Y 213.185,Z 493.669,A -85,B 0,C 180,E1 -30116.751,E2 -30116.751} C_VEL
LIN {X 0,Y 211.864,Z 507.972,A -85,B 0,C 180,E1 -30117.644,E2 -30117.644} C_VEL
LIN {X 0,Y 209.888,Z 521.684,A -85,B 0,C 180,E1 -30118.851,E2 -30118.851} C_VEL
LIN {X 0,Y 207.281,Z 534.881,A -85,B 0,C 180,E1 -30120.383,E2 -30120.383} C_VEL
LIN {X 0,Y 204.646,Z 546.759,A -85,B 0,C 180,E1 -30122.203,E2 -30122.203} C_VEL
LIN {X 0,Y 201.306,Z 558.808,A -85,B 0,C 180,E1 -30124.495,E2 -30124.495} C_VEL
LIN {X 0,Y 197.725,Z 569.655,A -85,B 0,C 180,E1 -30127.066,E2 -30127.066} C_VEL
LIN {X 0,Y 194.182,Z 579.62,A -85,B 0,C 180,E1 -30130.04,E2 -30130.04} C_VEL
LIN {X 0,Y 190.819,Z 588.708,A -85,B 0,C 180,E1 -30133.472,E2 -30133.472} C_VEL
LIN {X 0,Y 187.84,Z 596.252,A -85,B 0,C 180,E1 -30137.072,E2 -30137.072} C_VEL
LIN {X 0,Y 185.801,Z 601.508,A -85,B 0,C 180,E1 -30140.233,E2 -30140.233} C_VEL
LIN {X 0,Y 183.724,Z 607.062,A -85,B 0,C 180,E1 -30144.531,E2 -30144.531} C_VEL
LIN {X 0,Y 182.65,Z 610.218,A -85,B 0,C 180,E1 -30147.803,E2 -30147.803} C_VEL
LIN {X 0,Y 182.092,Z 613.175,A -85,B 0,C 180,E1 -30152.205,E2 -30152.205} C_VEL
LIN {X 0,Y 182.221,Z 614.819,A -85,B 0,C 180,E1 -30156.622,E2 -30156.622} C_VEL
LIN {X 0,Y 183.004,Z 615.185,A -85,B 0,C 180,E1 -30161.033,E2 -30161.033} C_VEL
LIN {X 0,Y 184.525,Z 614.264,A -85,B 0,C 180,E1 -30165.41,E2 -30165.41} C_VEL
LIN {X 0,Y 187.126,Z 611.995,A -85,B 0,C 180,E1 -30169.688,E2 -30169.688} C_VEL
LIN {X 0,Y 190.407,Z 608.35,A -85,B 0,C 180,E1 -30173.87,E2 -30173.87} C_VEL
LIN {X 0,Y 194.519,Z 603.161,A -85,B 0,C 180,E1 -30177.913,E2 -30177.913} C_VEL
LIN {X 0,Y 198.102,Z 598.156,A -85,B 0,C 180,E1 -30180.844,E2 -30180.844} C_VEL
LIN {X 0,Y 202.757,Z 590.965,A -85,B 0,C 180,E1 -30184.151,E2 -30184.151} C_VEL
LIN {X 0,Y 208.02,Z 581.966,A -85,B 0,C 180,E1 -30187.308,E2 -30187.308} C_VEL
LIN {X 0,Y 212.987,Z 572.511,A -85,B 0,C 180,E1 -30189.889,E2 -30189.889} C_VEL
LIN {X 0,Y 217.695,Z 561.776,A -85,B 0,C 180,E1 -30192.264,E2 -30192.264} C_VEL
LIN {X 0,Y 222.178,Z 550.336,A -85,B 0,C 180,E1 -30194.229,E2 -30194.229} C_VEL
LIN {X 0,Y 225.997,Z 538.865,A -85,B 0,C 180,E1 -30195.785,E2 -30195.785} C_VEL
LIN {X 0,Y 229.198,Z 526.347,A -85,B 0,C 180,E1 -30197.178,E2 -30197.178} C_VEL
LIN {X 0,Y 231.87,Z 512.637,A -85,B 0,C 180,E1 -30198.349,E2 -30198.349} C_VEL
LIN {X 0,Y 233.789,Z 498.651,A -85,B 0,C 180,E1 -30199.205,E2 -30199.205} C_VEL
LIN {X 0,Y 234.858,Z 484.227,A -85,B 0,C 180,E1 -30199.79,E2 -30199.79} C_VEL
LIN {X 0,Y 236.726,Z 452.363,A -85,B 0,C 180,E1 -30200.711,E2 -30200.711} C_VEL
LIN {X 0,Y 230.372,Z 439.912,A -85,B 0,C 180,E1 -30203.152,E2 -30203.152} C_VEL
LIN {X 0,Y 224.205,Z 429.325,A -85,B 0,C 180,E1 -30205.718,E2 -30205.718} C_VEL
LIN {X 0,Y 217.879,Z 419.279,A -85,B 0,C 180,E1 -30208.644,E2 -30208.644} C_VEL
LIN {X 0,Y 212.27,Z 411.295,A -85,B 0,C 180,E1 -30211.548,E2 -30211.548} C_VEL
LIN {X 0,Y 210.511,Z 408.924,A -85,B 0,C 180,E1 -30212.538,E2 -30212.538} C_VEL
LIN {X 0,Y 210.175,Z 409.237,A -85,B 0,C 180,E1 -30212.679,E2 -30212.679} C_VEL
LIN {X 0,Y 207.912,Z 414.774,A -85,B 0,C 180,E1 -30213.42,E2 -30213.42} C_VEL
LIN {X 0,Y 205.588,Z 419.053,A -85,B 0,C 180,E1 -30214.32,E2 -30214.32} C_VEL
LIN {X 0,Y 204.414,Z 420.582,A -85,B 0,C 180,E1 -30214.842,E2 -30214.842} C_VEL
LIN {X 0,Y 200.813,Z 434.189,A -85,B 0,C 180,E1 -30215.821,E2 -30215.821} C_VEL
LIN {X 0,Y 197.994,Z 443.074,A -85,B 0,C 180,E1 -30216.788,E2 -30216.788} C_VEL
LIN {X 0,Y 195.91,Z 447.933,A -85,B 0,C 180,E1 -30217.693,E2 -30217.693} C_VEL
LIN {X 0,Y 194.309,Z 450.038,A -85,B 0,C 180,E1 -30218.574,E2 -30218.574} C_VEL
LIN {X 0,Y 193.909,Z 450.319,A -85,B 0,C 180,E1 -30218.824,E2 -30218.824} C_VEL
LIN {X 0,Y 190.179,Z 465.492,A -85,B 0,C 180,E1 -30220.064,E2 -30220.064} C_VEL
LIN {X 0,Y 187.807,Z 473.462,A -85,B 0,C 180,E1 -30221.094,E2 -30221.094} C_VEL
LIN {X 0,Y 186.58,Z 476.137,A -85,B 0,C 180,E1 -30221.816,E2 -30221.816} C_VEL
LIN {X 0,Y 185.987,Z 476.144,A -85,B 0,C 180,E1 -30222.323,E2 -30222.323} C_VEL
LIN {X 0,Y 185.859,Z 474.134,A -85,B 0,C 180,E1 -30222.664,E2 -30222.664} C_VEL
LIN {X 0,Y 185.922,Z 472.102,A -85,B 0,C 180,E1 -30222.882,E2 -30222.882} C_VEL
LIN {X 0,Y 185.284,Z 495.185,A -85,B 0,C 180,E1 -30224.725,E2 -30224.725} C_VEL
LIN {X 0,Y 184.562,Z 510.658,A -85,B 0,C 180,E1 -30226.418,E2 -30226.418} C_VEL
LIN {X 0,Y 183.831,Z 527.033,A -85,B 0,C 180,E1 -30228.739,E2 -30228.739} C_VEL
LIN {X 0,Y 183.239,Z 539.365,A -85,B 0,C 180,E1 -30230.927,E2 -30230.927} C_VEL
LIN {X 0,Y 182.674,Z 552.078,A -85,B 0,C 180,E1 -30233.67,E2 -30233.67} C_VEL
LIN {X 0,Y 182.362,Z 565.098,A -85,B 0,C 180,E1 -30237.03,E2 -30237.03} C_VEL
LIN {X 0,Y 182.462,Z 574.872,A -85,B 0,C 180,E1 -30239.999,E2 -30239.999} C_VEL
LIN {X 0,Y 182.813,Z 585.451,A -85,B 0,C 180,E1 -30243.844,E2 -30243.844} C_VEL
LIN {X 0,Y 184.286,Z 595.599,A -85,B 0,C 180,E1 -30248.194,E2 -30248.194} C_VEL
LIN {X 0,Y 186.525,Z 603.038,A -85,B 0,C 180,E1 -30251.919,E2 -30251.919} C_VEL
LIN {X 0,Y 190.006,Z 610.113,A -85,B 0,C 180,E1 -30256.05,E2 -30256.05} C_VEL
LIN {X 0,Y 194.741,Z 615.85,A -85,B 0,C 180,E1 -30259.98,E2 -30259.98} C_VEL
LIN {X 0,Y 199.132,Z 619.366,A -85,B 0,C 180,E1 -30262.763,E2 -30262.763} C_VEL
LIN {X 0,Y 205.992,Z 622.932,A -85,B 0,C 180,E1 -30266.234,E2 -30266.234} C_VEL
LIN {X 0,Y 213.628,Z 625.303,A -85,B 0,C 180,E1 -30269.46,E2 -30269.46} C_VEL
LIN {X 0,Y 222.007,Z 626.506,A -85,B 0,C 180,E1 -30272.436,E2 -30272.436} C_VEL
LIN {X 0,Y 231.507,Z 626.482,A -85,B 0,C 180,E1 -30275.223,E2 -30275.223} C_VEL
LIN {X 0,Y 241.001,Z 625.338,A -85,B 0,C 180,E1 -30277.614,E2 -30277.614} C_VEL
LIN {X 0,Y 251.355,Z 622.923,A -85,B 0,C 180,E1 -30279.861,E2 -30279.861} C_VEL
LIN {X 0,Y 258.101,Z 620.774,A -85,B 0,C 180,E1 -30281.173,E2 -30281.173} C_VEL
LIN {X 0,Y 258.94,Z 620.638,A -85,B 0,C 180,E1 -30281.623,E2 -30281.623} C_VEL
LIN {X 0,Y 246.597,Z 626.789,A -85,B 0,C 180,E1 -30283.588,E2 -30283.588} C_VEL
LIN {X 0,Y 238.397,Z 630.326,A -85,B 0,C 180,E1 -30285.157,E2 -30285.157} C_VEL
LIN {X 0,Y 226.987,Z 634.412,A -85,B 0,C 180,E1 -30287.782,E2 -30287.782} C_VEL
LIN {X 0,Y 218.574,Z 636.737,A -85,B 0,C 180,E1 -30290.139,E2 -30290.139} C_VEL
LIN {X 0,Y 210.852,Z 638.343,A -85,B 0,C 180,E1 -30292.785,E2 -30292.785} C_VEL
LIN {X 0,Y 206.944,Z 638.782,A -85,B 0,C 180,E1 -30293.998,E2 -30293.998} C_VEL
LIN {X 0,Y 199.518,Z 638.691,A -85,B 0,C 180,E1 -30295.854,E2 -30295.854} C_VEL
LIN {X 0,Y 192.587,Z 637.988,A -85,B 0,C 180,E1 -30297.899,E2 -30297.899} C_VEL
LIN {X 0,Y 189.524,Z 637.488,A -85,B 0,C 180,E1 -30299.397,E2 -30299.397} C_VEL
LIN {X 0,Y 184.738,Z 636.379,A -85,B 0,C 180,E1 -30303.164,E2 -30303.164} C_VEL
LIN {X 0,Y 179.958,Z 642.471,A -85,B 0,C 180,E1 -30307.093,E2 -30307.093} C_VEL
LIN {X 0,Y 176.448,Z 647.358,A -85,B 0,C 180,E1 -30311.483,E2 -30311.483} C_VEL
LIN {X 0,Y 174.315,Z 650.802,A -85,B 0,C 180,E1 -30316.048,E2 -30316.048} C_VEL
LIN {X 0,Y 173.885,Z 652.948,A -85,B 0,C 180,E1 -30320.727,E2 -30320.727} C_VEL
LIN {X 0,Y 175.069,Z 653.846,A -85,B 0,C 180,E1 -30325.41,E2 -30325.41} C_VEL
LIN {X 0,Y 177.065,Z 653.828,A -85,B 0,C 180,E1 -30328.795,E2 -30328.795} C_VEL
LIN {X 0,Y 177.102,Z 662.227,A -85,B 0,C 180,E1 -30331.699,E2 -30331.699} C_VEL
LIN {X 0,Y 176.844,Z 669.063,A -85,B 0,C 180,E1 -30334.543,E2 -30334.543} C_VEL
LIN {X 0,Y 176.448,Z 676.917,A -85,B 0,C 180,E1 -30338.56,E2 -30338.56} C_VEL
LIN {X 0,Y 176.754,Z 683.455,A -85,B 0,C 180,E1 -30342.589,E2 -30342.589} C_VEL
LIN {X 0,Y 178.554,Z 689.725,A -85,B 0,C 180,E1 -30347.11,E2 -30347.11} C_VEL
LIN {X 0,Y 181.729,Z 694.802,A -85,B 0,C 180,E1 -30351.479,E2 -30351.479} C_VEL
LIN {X 0,Y 187.691,Z 699.698,A -85,B 0,C 180,E1 -30356.604,E2 -30356.604} C_VEL
LIN {X 0,Y 193.687,Z 702.424,A -85,B 0,C 180,E1 -30360.417,E2 -30360.417} C_VEL
LIN {X 0,Y 200.964,Z 704.192,A -85,B 0,C 180,E1 -30363.894,E2 -30363.894} C_VEL
LIN {X 0,Y 209.323,Z 705.003,A -85,B 0,C 180,E1 -30367.036,E2 -30367.036} C_VEL
LIN {X 0,Y 218.585,Z 704.826,A -85,B 0,C 180,E1 -30369.858,E2 -30369.858} C_VEL
LIN {X 0,Y 228.558,Z 703.633,A -85,B 0,C 180,E1 -30372.393,E2 -30372.393} C_VEL
LIN {X 0,Y 240.324,Z 701.095,A -85,B 0,C 180,E1 -30374.829,E2 -30374.829} C_VEL
LIN {X 0,Y 239.613,Z 701.262,A -85,B 0,C 180,E1 -30375.447,E2 -30375.447} C_VEL
LIN {X 0,Y 228.909,Z 703.512,A -85,B 0,C 180,E1 -30377.687,E2 -30377.687} C_VEL
LIN {X 0,Y 217.82,Z 704.766,A -85,B 0,C 180,E1 -30380.513,E2 -30380.513} C_VEL
LIN {X 0,Y 209.683,Z 704.831,A -85,B 0,C 180,E1 -30383.038,E2 -30383.038} C_VEL
LIN {X 0,Y 201.385,Z 704.004,A -85,B 0,C 180,E1 -30386.186,E2 -30386.186} C_VEL
LIN {X 0,Y 193.994,Z 702.199,A -85,B 0,C 180,E1 -30389.636,E2 -30389.636} C_VEL
LIN {X 0,Y 187.773,Z 699.337,A -85,B 0,C 180,E1 -30393.542,E2 -30393.542} C_VEL
LIN {X 0,Y 181.858,Z 694.48,A -85,B 0,C 180,E1 -30398.537,E2 -30398.537} C_VEL
LIN {X 0,Y 178.606,Z 689.361,A -85,B 0,C 180,E1 -30402.895,E2 -30402.895} C_VEL
LIN {X 0,Y 176.715,Z 683.052,A -85,B 0,C 180,E1 -30407.409,E2 -30407.409} C_VEL
LIN {X 0,Y 176.299,Z 676.478,A -85,B 0,C 180,E1 -30411.432,E2 -30411.432} C_VEL
LIN {X 0,Y 176.658,Z 667.361,A -85,B 0,C 180,E1 -30416.022,E2 -30416.022} C_VEL
LIN {X 0,Y 176.911,Z 660.295,A -85,B 0,C 180,E1 -30418.866,E2 -30418.866} C_VEL
LIN {X 0,Y 176.93,Z 651.918,A -85,B 0,C 180,E1 -30421.702,E2 -30421.702} C_VEL
LIN {X 0,Y 177.027,Z 640.521,A -85,B 0,C 180,E1 -30424.899,E2 -30424.899} C_VEL
LIN {X 0,Y 177.338,Z 626.597,A -85,B 0,C 180,E1 -30428.099,E2 -30428.099} C_VEL
LIN {X 0,Y 177.748,Z 612.14,A -85,B 0,C 180,E1 -30430.732,E2 -30430.732} C_VEL
LIN {X 0,Y 178.379,Z 597.197,A -85,B 0,C 180,E1 -30432.905,E2 -30432.905} C_VEL
LIN {X 0,Y 178.862,Z 580.931,A -85,B 0,C 180,E1 -30434.675,E2 -30434.675} C_VEL
LIN {X 0,Y 179.878,Z 537.62,A -85,B 0,C 180,E1 -30438.225,E2 -30438.225} C_VEL
LIN {X 0,Y 181.759,Z 481.326,A -85,B 0,C 180,E1 -30442.622,E2 -30442.622} C_VEL
LIN {X 0,Y 179.843,Z 451.312,A -85,B 0,C 180,E1 -30444.829,E2 -30444.829} C_VEL
LIN {X 0,Y 179.717,Z 439.56,A -85,B 0,C 180,E1 -30445.727,E2 -30445.727} C_VEL
LIN {X 0,Y 183.212,Z 412.821,A -85,B 0,C 180,E1 -30452.361,E2 -30452.361} C_VEL
LIN {X 0,Y 182.957,Z 409.778,A -85,B 0,C 180,E1 -30453.126,E2 -30453.126} C_VEL
LIN {X 0,Y 178.598,Z 389.913,A -85,B 0,C 180,E1 -30458.337,E2 -30458.337} C_VEL
LIN {X 0,Y 176.936,Z 382.476,A -85,B 0,C 180,E1 -30460.363,E2 -30460.363} C_VEL
LIN {X 0,Y 177.824,Z 384.259,A -85,B 0,C 180,E1 -30460.883,E2 -30460.883} C_VEL
LIN {X 0,Y 179.425,Z 384.805,A -85,B 0,C 180,E1 -30461.58,E2 -30461.58} C_VEL
LIN {X 0,Y 181.292,Z 384.858,A -85,B 0,C 180,E1 -30462.328,E2 -30462.328} C_VEL
LIN {X 0,Y 183.006,Z 386.855,A -85,B 0,C 180,E1 -30463.109,E2 -30463.109} C_VEL
LIN {X 0,Y 185.741,Z 390.595,A -85,B 0,C 180,E1 -30464.333,E2 -30464.333} C_VEL
LIN {X 0,Y 191.877,Z 399.736,A -85,B 0,C 180,E1 -30466.896,E2 -30466.896} C_VEL
LIN {X 0,Y 198.505,Z 410.382,A -85,B 0,C 180,E1 -30469.407,E2 -30469.407} C_VEL
LIN {X 0,Y 205.422,Z 423.127,A -85,B 0,C 180,E1 -30471.833,E2 -30471.833} C_VEL
LIN {X 0,Y 210.464,Z 433.706,A -85,B 0,C 180,E1 -30473.505,E2 -30473.505} C_VEL
LIN {X 0,Y 207.83,Z 488.794,A -85,B 0,C 180,E1 -30475.338,E2 -30475.338} C_VEL
LIN {X 0,Y 206.867,Z 502.794,A -85,B 0,C 180,E1 -30476.109,E2 -30476.109} C_VEL
LIN {X 0,Y 205.092,Z 516.462,A -85,B 0,C 180,E1 -30477.168,E2 -30477.168} C_VEL
LIN {X 0,Y 202.753,Z 529.249,A -85,B 0,C 180,E1 -30478.499,E2 -30478.499} C_VEL
LIN {X 0,Y 200.183,Z 540.95,A -85,B 0,C 180,E1 -30480.092,E2 -30480.092} C_VEL
LIN {X 0,Y 197.062,Z 553.118,A -85,B 0,C 180,E1 -30482.192,E2 -30482.192} C_VEL
LIN {X 0,Y 193.617,Z 564.171,A -85,B 0,C 180,E1 -30484.558,E2 -30484.558} C_VEL
LIN {X 0,Y 190.157,Z 573.899,A -85,B 0,C 180,E1 -30487.132,E2 -30487.132} C_VEL
LIN {X 0,Y 186.61,Z 583.323,A -85,B 0,C 180,E1 -30490.256,E2 -30490.256} C_VEL
LIN {X 0,Y 183.65,Z 590.898,A -85,B 0,C 180,E1 -30493.379,E2 -30493.379} C_VEL
LIN {X 0,Y 180.977,Z 597.207,A -85,B 0,C 180,E1 -30496.572,E2 -30496.572} C_VEL
LIN {X 0,Y 178.867,Z 602.424,A -85,B 0,C 180,E1 -30499.851,E2 -30499.851} C_VEL
LIN {X 0,Y 176.693,Z 607.946,A -85,B 0,C 180,E1 -30504.313,E2 -30504.313} C_VEL
LIN {X 0,Y 175.608,Z 611.068,A -85,B 0,C 180,E1 -30507.714,E2 -30507.714} C_VEL
LIN {X 0,Y 175.034,Z 613.995,A -85,B 0,C 180,E1 -30512.294,E2 -30512.294} C_VEL
LIN {X 0,Y 175.18,Z 615.612,A -85,B 0,C 180,E1 -30516.89,E2 -30516.89} C_VEL
LIN {X 0,Y 176.041,Z 615.949,A -85,B 0,C 180,E1 -30521.476,E2 -30521.476} C_VEL
LIN {X 0,Y 177.691,Z 614.998,A -85,B 0,C 180,E1 -30526.018,E2 -30526.018} C_VEL
LIN {X 0,Y 180.474,Z 612.696,A -85,B 0,C 180,E1 -30530.445,E2 -30530.445} C_VEL
LIN {X 0,Y 183.94,Z 609.02,A -85,B 0,C 180,E1 -30534.764,E2 -30534.764} C_VEL
LIN {X 0,Y 188.27,Z 603.781,A -85,B 0,C 180,E1 -30538.925,E2 -30538.925} C_VEL
LIN {X 0,Y 192.047,Z 598.756,A -85,B 0,C 180,E1 -30541.928,E2 -30541.928} C_VEL
LIN {X 0,Y 196.904,Z 591.519,A -85,B 0,C 180,E1 -30545.315,E2 -30545.315} C_VEL
LIN {X 0,Y 201.604,Z 583.898,A -85,B 0,C 180,E1 -30548.076,E2 -30548.076} C_VEL
LIN {X 0,Y 206.73,Z 574.7,A -85,B 0,C 180,E1 -30550.71,E2 -30550.71} C_VEL
LIN {X 0,Y 211.538,Z 564.316,A -85,B 0,C 180,E1 -30553.129,E2 -30553.129} C_VEL
LIN {X 0,Y 216.155,Z 553.184,A -85,B 0,C 180,E1 -30555.142,E2 -30555.142} C_VEL
LIN {X 0,Y 220.612,Z 540.609,A -85,B 0,C 180,E1 -30556.908,E2 -30556.908} C_VEL
LIN {X 0,Y 223.924,Z 528.346,A -85,B 0,C 180,E1 -30558.316,E2 -30558.316} C_VEL
LIN {X 0,Y 226.769,Z 514.636,A -85,B 0,C 180,E1 -30559.527,E2 -30559.527} C_VEL
LIN {X 0,Y 228.787,Z 501.081,A -85,B 0,C 180,E1 -30560.393,E2 -30560.393} C_VEL
LIN {X 0,Y 230.024,Z 486.901,A -85,B 0,C 180,E1 -30561.007,E2 -30561.007} C_VEL
LIN {X 0,Y 231.896,Z 455.084,A -85,B 0,C 180,E1 -30561.962,E2 -30561.962} C_VEL
LIN {X 0,Y 226.144,Z 443.715,A -85,B 0,C 180,E1 -30564.311,E2 -30564.311} C_VEL
LIN {X 0,Y 220.012,Z 433.048,A -85,B 0,C 180,E1 -30567.029,E2 -30567.029} C_VEL
LIN {X 0,Y 214.293,Z 423.912,A -85,B 0,C 180,E1 -30569.847,E2 -30569.847} C_VEL
LIN {X 0,Y 210.802,Z 418.747,A -85,B 0,C 180,E1 -30571.738,E2 -30571.738} C_VEL
LIN {X 0,Y 210.372,Z 418.662,A -85,B 0,C 180,E1 -30571.946,E2 -30571.946} C_VEL
LIN {X 0,Y 207.848,Z 423.4,A -85,B 0,C 180,E1 -30572.845,E2 -30572.845} C_VEL
LIN {X 0,Y 206.797,Z 424.925,A -85,B 0,C 180,E1 -30573.265,E2 -30573.265} C_VEL
LIN {X 0,Y 202.89,Z 438.821,A -85,B 0,C 180,E1 -30574.298,E2 -30574.298} C_VEL
LIN {X 0,Y 199.819,Z 447.806,A -85,B 0,C 180,E1 -30575.317,E2 -30575.317} C_VEL
LIN {X 0,Y 197.37,Z 453.089,A -85,B 0,C 180,E1 -30576.336,E2 -30576.336} C_VEL
LIN {X 0,Y 195.572,Z 455.858,A -85,B 0,C 180,E1 -30577.221,E2 -30577.221} C_VEL
LIN {X 0,Y 192.115,Z 469.224,A -85,B 0,C 180,E1 -30578.317,E2 -30578.317} C_VEL
LIN {X 0,Y 189.514,Z 477.441,A -85,B 0,C 180,E1 -30579.382,E2 -30579.382} C_VEL
LIN {X 0,Y 187.607,Z 481.546,A -85,B 0,C 180,E1 -30580.41,E2 -30580.41} C_VEL
LIN {X 0,Y 186.344,Z 483.019,A -85,B 0,C 180,E1 -30581.264,E2 -30581.264} C_VEL
LIN {X 0,Y 186.093,Z 483.172,A -85,B 0,C 180,E1 -30581.454,E2 -30581.454} C_VEL
LIN {X 0,Y 183.179,Z 495.527,A -85,B 0,C 180,E1 -30582.574,E2 -30582.574} C_VEL
LIN {X 0,Y 180.888,Z 503.156,A -85,B 0,C 180,E1 -30583.622,E2 -30583.622} C_VEL
LIN {X 0,Y 179.067,Z 507.381,A -85,B 0,C 180,E1 -30584.617,E2 -30584.617} C_VEL
LIN {X 0,Y 178.089,Z 508.978,A -85,B 0,C 180,E1 -30585.333,E2 -30585.333} C_VEL
LIN {X 0,Y 177.671,Z 508.977,A -85,B 0,C 180,E1 -30585.808,E2 -30585.808} C_VEL
LIN {X 0,Y 177.603,Z 508.096,A -85,B 0,C 180,E1 -30586.093,E2 -30586.093} C_VEL
LIN {X 0,Y 177.809,Z 506.076,A -85,B 0,C 180,E1 -30586.328,E2 -30586.328} C_VEL
LIN {X 0,Y 177.077,Z 524.044,A -85,B 0,C 180,E1 -30588.881,E2 -30588.881} C_VEL
LIN {X 0,Y 176.417,Z 538.304,A -85,B 0,C 180,E1 -30591.437,E2 -30591.437} C_VEL
LIN {X 0,Y 175.845,Z 551.833,A -85,B 0,C 180,E1 -30594.399,E2 -30594.399} C_VEL
LIN {X 0,Y 175.597,Z 564.362,A -85,B 0,C 180,E1 -30597.713,E2 -30597.713} C_VEL
LIN {X 0,Y 175.742,Z 575.169,A -85,B 0,C 180,E1 -30601.141,E2 -30601.141} C_VEL
LIN {X 0,Y 176.422,Z 586.902,A -85,B 0,C 180,E1 -30605.554,E2 -30605.554} C_VEL
LIN {X 0,Y 178.12,Z 596.3,A -85,B 0,C 180,E1 -30609.761,E2 -30609.761} C_VEL
LIN {X 0,Y 181.374,Z 605.445,A -85,B 0,C 180,E1 -30614.537,E2 -30614.537} C_VEL
LIN {X 0,Y 185.512,Z 612.25,A -85,B 0,C 180,E1 -30618.719,E2 -30618.719} C_VEL
LIN {X 0,Y 191.025,Z 617.814,A -85,B 0,C 180,E1 -30622.644,E2 -30622.644} C_VEL
LIN {X 0,Y 196.017,Z 621.13,A -85,B 0,C 180,E1 -30625.391,E2 -30625.391} C_VEL
LIN {X 0,Y 203.438,Z 624.53,A -85,B 0,C 180,E1 -30628.817,E2 -30628.817} C_VEL
LIN {X 0,Y 211.689,Z 626.754,A -85,B 0,C 180,E1 -30631.965,E2 -30631.965} C_VEL
LIN {X 0,Y 220.72,Z 627.815,A -85,B 0,C 180,E1 -30634.835,E2 -30634.835} C_VEL
LIN {X 0,Y 230.441,Z 627.714,A -85,B 0,C 180,E1 -30637.439,E2 -30637.439} C_VEL
LIN {X 0,Y 240.784,Z 626.412,A -85,B 0,C 180,E1 -30639.79,E2 -30639.79} C_VEL
LIN {X 0,Y 247.111,Z 625.09,A -85,B 0,C 180,E1 -30641.067,E2 -30641.067} C_VEL
LIN {X 0,Y 246.287,Z 625.685,A -85,B 0,C 180,E1 -30641.617,E2 -30641.617} C_VEL
LIN {X 0,Y 233.413,Z 630.691,A -85,B 0,C 180,E1 -30643.928,E2 -30643.928} C_VEL
LIN {X 0,Y 222.913,Z 633.922,A -85,B 0,C 180,E1 -30646.267,E2 -30646.267} C_VEL
LIN {X 0,Y 213.2,Z 636.204,A -85,B 0,C 180,E1 -30648.922,E2 -30648.922} C_VEL
LIN {X 0,Y 204.428,Z 637.578,A -85,B 0,C 180,E1 -30651.921,E2 -30651.921} C_VEL
LIN {X 0,Y 196.796,Z 638.038,A -85,B 0,C 180,E1 -30655.285,E2 -30655.285} C_VEL
LIN {X 0,Y 189.524,Z 637.488,A -85,B 0,C 180,E1 -30659.397,E2 -30659.397} C_VEL
LIN {X 0,Y 186.582,Z 637.454,A -85,B 0,C 180,E1 -30660.944,E2 -30660.944} C_VEL
LIN {X 0,Y 182.944,Z 638.081,A -85,B 0,C 180,E1 -30662.378,E2 -30662.378} C_VEL
LIN {X 0,Y 177.891,Z 639.711,A -85,B 0,C 180,E1 -30664.259,E2 -30664.259} C_VEL
LIN {X 0,Y 173.632,Z 642.017,A -85,B 0,C 180,E1 -30666.315,E2 -30666.315} C_VEL
LIN {X 0,Y 172.222,Z 643.339,A -85,B 0,C 180,E1 -30667.46,E2 -30667.46} C_VEL
LIN {X 0,Y 169.71,Z 646.666,A -85,B 0,C 180,E1 -30670.72,E2 -30670.72} C_VEL
LIN {X 0,Y 167.389,Z 650.072,A -85,B 0,C 180,E1 -30675.459,E2 -30675.459} C_VEL
LIN {X 0,Y 166.792,Z 652.186,A -85,B 0,C 180,E1 -30680.329,E2 -30680.329} C_VEL
LIN {X 0,Y 167.873,Z 653.054,A -85,B 0,C 180,E1 -30685.213,E2 -30685.213} C_VEL
LIN {X 0,Y 170.582,Z 652.895,A -85,B 0,C 180,E1 -30689.779,E2 -30689.779} C_VEL
LIN {X 0,Y 170.612,Z 660.161,A -85,B 0,C 180,E1 -30692.353,E2 -30692.353} C_VEL
LIN {X 0,Y 170.318,Z 667.686,A -85,B 0,C 180,E1 -30695.574,E2 -30695.574} C_VEL
LIN {X 0,Y 170.014,Z 676.154,A -85,B 0,C 180,E1 -30700.084,E2 -30700.084} C_VEL
LIN {X 0,Y 171.029,Z 684.356,A -85,B 0,C 180,E1 -30705.438,E2 -30705.438} C_VEL
LIN {X 0,Y 173.524,Z 690.361,A -85,B 0,C 180,E1 -30710.066,E2 -30710.066} C_VEL
LIN {X 0,Y 177.957,Z 695.618,A -85,B 0,C 180,E1 -30714.789,E2 -30714.789} C_VEL
LIN {X 0,Y 184.463,Z 699.949,A -85,B 0,C 180,E1 -30719.58,E2 -30719.58} C_VEL
LIN {X 0,Y 191.255,Z 702.592,A -85,B 0,C 180,E1 -30723.323,E2 -30723.323} C_VEL
LIN {X 0,Y 199.309,Z 704.269,A -85,B 0,C 180,E1 -30726.687,E2 -30726.687} C_VEL
LIN {X 0,Y 208.373,Z 704.993,A -85,B 0,C 180,E1 -30729.694,E2 -30729.694} C_VEL
LIN {X 0,Y 218.18,Z 704.747,A -85,B 0,C 180,E1 -30732.391,E2 -30732.391} C_VEL
LIN {X 0,Y 228.743,Z 703.51,A -85,B 0,C 180,E1 -30734.772,E2 -30734.772} C_VEL
LIN {X 0,Y 229.077,Z 703.444,A -85,B 0,C 180,E1 -30735.311,E2 -30735.311} C_VEL
LIN {X 0,Y 218.509,Z 704.658,A -85,B 0,C 180,E1 -30737.689,E2 -30737.689} C_VEL
LIN {X 0,Y 208.662,Z 704.879,A -85,B 0,C 180,E1 -30740.373,E2 -30740.373} C_VEL
LIN {X 0,Y 199.701,Z 704.139,A -85,B 0,C 180,E1 -30743.397,E2 -30743.397} C_VEL
LIN {X 0,Y 191.613,Z 702.426,A -85,B 0,C 180,E1 -30746.748,E2 -30746.748} C_VEL
LIN {X 0,Y 184.714,Z 699.735,A -85,B 0,C 180,E1 -30750.465,E2 -30750.465} C_VEL
LIN {X 0,Y 177.782,Z 695.039,A -85,B 0,C 180,E1 -30755.564,E2 -30755.564} C_VEL
LIN {X 0,Y 173.636,Z 690.058,A -85,B 0,C 180,E1 -30759.948,E2 -30759.948} C_VEL
LIN {X 0,Y 171.018,Z 684,A -85,B 0,C 180,E1 -30764.561,E2 -30764.561} C_VEL
LIN {X 0,Y 169.907,Z 675.759,A -85,B 0,C 180,E1 -30769.91,E2 -30769.91} C_VEL
LIN {X 0,Y 170.088,Z 666.826,A -85,B 0,C 180,E1 -30774.612,E2 -30774.612} C_VEL
LIN {X 0,Y 170.375,Z 659.758,A -85,B 0,C 180,E1 -30777.644,E2 -30777.644} C_VEL
LIN {X 0,Y 170.417,Z 651.464,A -85,B 0,C 180,E1 -30780.589,E2 -30780.589} C_VEL
LIN {X 0,Y 170.407,Z 639.341,A -85,B 0,C 180,E1 -30784.126,E2 -30784.126} C_VEL
LIN {X 0,Y 170.614,Z 627.033,A -85,B 0,C 180,E1 -30787.075,E2 -30787.075} C_VEL
LIN {X 0,Y 170.925,Z 613.284,A -85,B 0,C 180,E1 -30789.731,E2 -30789.731} C_VEL
LIN {X 0,Y 171.483,Z 598.138,A -85,B 0,C 180,E1 -30792.084,E2 -30792.084} C_VEL
LIN {X 0,Y 171.937,Z 583.299,A -85,B 0,C 180,E1 -30793.848,E2 -30793.848} C_VEL
LIN {X 0,Y 172.592,Z 552.066,A -85,B 0,C 180,E1 -30796.581,E2 -30796.581} C_VEL
LIN {X 0,Y 174.685,Z 481.282,A -85,B 0,C 180,E1 -30802.433,E2 -30802.433} C_VEL
LIN {X 0,Y 172.753,Z 451.396,A -85,B 0,C 180,E1 -30804.717,E2 -30804.717} C_VEL
LIN {X 0,Y 172.644,Z 439.432,A -85,B 0,C 180,E1 -30805.698,E2 -30805.698} C_VEL
LIN {X 0,Y 176.107,Z 413.072,A -85,B 0,C 180,E1 -30812.477,E2 -30812.477} C_VEL
LIN {X 0,Y 175.798,Z 410.278,A -85,B 0,C 180,E1 -30813.205,E2 -30813.205} C_VEL
LIN {X 0,Y 171.541,Z 390.75,A -85,B 0,C 180,E1 -30818.518,E2 -30818.518} C_VEL
LIN {X 0,Y 172.335,Z 392.543,A -85,B 0,C 180,E1 -30819.018,E2 -30819.018} C_VEL
LIN {X 0,Y 172.86,Z 392.903,A -85,B 0,C 180,E1 -30819.285,E2 -30819.285} C_VEL
LIN {X 0,Y 174.871,Z 392.786,A -85,B 0,C 180,E1 -30820.179,E2 -30820.179} C_VEL
LIN {X 0,Y 176.323,Z 391.778,A -85,B 0,C 180,E1 -30820.74,E2 -30820.74} C_VEL
LIN {X 0,Y 179.497,Z 392.111,A -85,B 0,C 180,E1 -30822.07,E2 -30822.07} C_VEL
LIN {X 0,Y 185.908,Z 401.498,A -85,B 0,C 180,E1 -30825.018,E2 -30825.018} C_VEL
LIN {X 0,Y 192.734,Z 412.387,A -85,B 0,C 180,E1 -30827.829,E2 -30827.829} C_VEL
LIN {X 0,Y 199.312,Z 424.285,A -85,B 0,C 180,E1 -30830.308,E2 -30830.308} C_VEL
LIN {X 0,Y 204.963,Z 435.999,A -85,B 0,C 180,E1 -30832.308,E2 -30832.308} C_VEL
LIN {X 0,Y 202.305,Z 488.864,A -85,B 0,C 180,E1 -30834.096,E2 -30834.096} C_VEL
LIN {X 0,Y 201.277,Z 503.138,A -85,B 0,C 180,E1 -30834.88,E2 -30834.88} C_VEL
LIN {X 0,Y 199.451,Z 516.92,A -85,B 0,C 180,E1 -30835.965,E2 -30835.965} C_VEL
LIN {X 0,Y 196.811,Z 530.753,A -85,B 0,C 180,E1 -30837.433,E2 -30837.433} C_VEL
LIN {X 0,Y 194.167,Z 542.299,A -85,B 0,C 180,E1 -30839.066,E2 -30839.066} C_VEL
LIN {X 0,Y 190.881,Z 554.351,A -85,B 0,C 180,E1 -30841.209,E2 -30841.209} C_VEL
LIN {X 0,Y 187.662,Z 564.292,A -85,B 0,C 180,E1 -30843.391,E2 -30843.391} C_VEL
LIN {X 0,Y 183.703,Z 574.978,A -85,B 0,C 180,E1 -30846.281,E2 -30846.281} C_VEL
LIN {X 0,Y 179.997,Z 584.342,A -85,B 0,C 180,E1 -30849.499,E2 -30849.499} C_VEL
LIN {X 0,Y 176.917,Z 591.878,A -85,B 0,C 180,E1 -30852.727,E2 -30852.727} C_VEL
LIN {X 0,Y 174.13,Z 598.162,A -85,B 0,C 180,E1 -30856.034,E2 -30856.034} C_VEL
LIN {X 0,Y 171.944,Z 603.34,A -85,B 0,C 180,E1 -30859.437,E2 -30859.437} C_VEL
LIN {X 0,Y 169.668,Z 608.83,A -85,B 0,C 180,E1 -30864.076,E2 -30864.076} C_VEL
LIN {X 0,Y 168.568,Z 611.917,A -85,B 0,C 180,E1 -30867.619,E2 -30867.619} C_VEL
LIN {X 0,Y 167.978,Z 614.815,A -85,B 0,C 180,E1 -30872.39,E2 -30872.39} C_VEL
LIN {X 0,Y 168.158,Z 616.403,A -85,B 0,C 180,E1 -30877.179,E2 -30877.179} C_VEL
LIN {X 0,Y 169.1,Z 616.712,A -85,B 0,C 180,E1 -30881.953,E2 -30881.953} C_VEL
LIN {X 0,Y 170.881,Z 615.731,A -85,B 0,C 180,E1 -30886.675,E2 -30886.675} C_VEL
LIN {X 0,Y 173.836,Z 613.4,A -85,B 0,C 180,E1 -30891.263,E2 -30891.263} C_VEL
LIN {X 0,Y 177.514,Z 609.686,A -85,B 0,C 180,E1 -30895.725,E2 -30895.725} C_VEL
LIN {X 0,Y 182.067,Z 604.402,A -85,B 0,C 180,E1 -30900.009,E2 -30900.009} C_VEL
LIN {X 0,Y 186.068,Z 599.354,A -85,B 0,C 180,E1 -30903.083,E2 -30903.083} C_VEL
LIN {X 0,Y 191.14,Z 592.064,A -85,B 0,C 180,E1 -30906.548,E2 -30906.548} C_VEL
LIN {X 0,Y 196.043,Z 584.407,A -85,B 0,C 180,E1 -30909.361,E2 -30909.361} C_VEL
LIN {X 0,Y 201.388,Z 575.14,A -85,B 0,C 180,E1 -30912.032,E2 -30912.032} C_VEL
LIN {X 0,Y 206.173,Z 565.215,A -85,B 0,C 180,E1 -30914.37,E2 -30914.37} C_VEL
LIN {X 0,Y 211.201,Z 553.465,A -85,B 0,C 180,E1 -30916.51,E2 -30916.51} C_VEL
LIN {X 0,Y 215.797,Z 540.781,A -85,B 0,C 180,E1 -30918.293,E2 -30918.293} C_VEL
LIN {X 0,Y 219.248,Z 528.362,A -85,B 0,C 180,E1 -30919.708,E2 -30919.708} C_VEL
LIN {X 0,Y 222.096,Z 514.913,A -85,B 0,C 180,E1 -30920.893,E2 -30920.893} C_VEL
LIN {X 0,Y 224.2,Z 501.177,A -85,B 0,C 180,E1 -30921.761,E2 -30921.761} C_VEL
LIN {X 0,Y 225.465,Z 486.384,A -85,B 0,C 180,E1 -30922.393,E2 -30922.393} C_VEL
LIN {X 0,Y 227.167,Z 457.822,A -85,B 0,C 180,E1 -30923.272,E2 -30923.272} C_VEL
LIN {X 0,Y 221.948,Z 447.49,A -85,B 0,C 180,E1 -30925.539,E2 -30925.539} C_VEL
LIN {X 0,Y 215.874,Z 436.694,A -85,B 0,C 180,E1 -30928.42,E2 -30928.42} C_VEL
LIN {X 0,Y 210.281,Z 427.656,A -85,B 0,C 180,E1 -30931.39,E2 -30931.39} C_VEL
LIN {X 0,Y 209.359,Z 429.025,A -85,B 0,C 180,E1 -30931.73,E2 -30931.73} C_VEL
LIN {X 0,Y 205.46,Z 442.355,A -85,B 0,C 180,E1 -30932.707,E2 -30932.707} C_VEL
LIN {X 0,Y 202.151,Z 451.605,A -85,B 0,C 180,E1 -30933.743,E2 -30933.743} C_VEL
LIN {X 0,Y 199.317,Z 457.564,A -85,B 0,C 180,E1 -30934.839,E2 -30934.839} C_VEL
LIN {X 0,Y 197.7,Z 460.209,A -85,B 0,C 180,E1 -30935.559,E2 -30935.559} C_VEL
LIN {X 0,Y 194.1,Z 473.345,A -85,B 0,C 180,E1 -30936.654,E2 -30936.654} C_VEL
LIN {X 0,Y 191.418,Z 481.332,A -85,B 0,C 180,E1 -30937.689,E2 -30937.689} C_VEL
LIN {X 0,Y 188.988,Z 486.473,A -85,B 0,C 180,E1 -30938.892,E2 -30938.892} C_VEL
LIN {X 0,Y 187.487,Z 488.831,A -85,B 0,C 180,E1 -30939.765,E2 -30939.765} C_VEL
LIN {X 0,Y 184.775,Z 499.274,A -85,B 0,C 180,E1 -30940.728,E2 -30940.728} C_VEL
LIN {X 0,Y 181.996,Z 507.231,A -85,B 0,C 180,E1 -30941.817,E2 -30941.817} C_VEL
LIN {X 0,Y 179.553,Z 512.311,A -85,B 0,C 180,E1 -30942.987,E2 -30942.987} C_VEL
LIN {X 0,Y 177.815,Z 514.978,A -85,B 0,C 180,E1 -30944.067,E2 -30944.067} C_VEL
LIN {X 0,Y 176.528,Z 515.981,A -85,B 0,C 180,E1 -30945.2,E2 -30945.2} C_VEL
LIN {X 0,Y 173.75,Z 522.253,A -85,B 0,C 180,E1 -30946.369,E2 -30946.369} C_VEL
LIN {X 0,Y 172.527,Z 524.677,A -85,B 0,C 180,E1 -30947.005,E2 -30947.005} C_VEL
LIN {X 0,Y 170.777,Z 527.431,A -85,B 0,C 180,E1 -30948.165,E2 -30948.165} C_VEL
LIN {X 0,Y 169.804,Z 528.216,A -85,B 0,C 180,E1 -30949.302,E2 -30949.302} C_VEL
LIN {X 0,Y 170.058,Z 526.512,A -85,B 0,C 180,E1 -30949.993,E2 -30949.993} C_VEL
LIN {X 0,Y 169.457,Z 541.033,A -85,B 0,C 180,E1 -30952.767,E2 -30952.767} C_VEL
LIN {X 0,Y 168.995,Z 553.884,A -85,B 0,C 180,E1 -30955.815,E2 -30955.815} C_VEL
LIN {X 0,Y 168.942,Z 566.527,A -85,B 0,C 180,E1 -30959.405,E2 -30959.405} C_VEL
LIN {X 0,Y 169.155,Z 577.095,A -85,B 0,C 180,E1 -30962.966,E2 -30962.966} C_VEL
LIN {X 0,Y 170.04,Z 587.492,A -85,B 0,C 180,E1 -30967.098,E2 -30967.098} C_VEL
LIN {X 0,Y 172.252,Z 597.508,A -85,B 0,C 180,E1 -30971.731,E2 -30971.731} C_VEL
LIN {X 0,Y 175.581,Z 605.828,A -85,B 0,C 180,E1 -30976.215,E2 -30976.215} C_VEL
LIN {X 0,Y 180.125,Z 612.762,A -85,B 0,C 180,E1 -30980.485,E2 -30980.485} C_VEL
LIN {X 0,Y 186.118,Z 618.414,A -85,B 0,C 180,E1 -30984.455,E2 -30984.455} C_VEL
LIN {X 0,Y 193.333,Z 622.87,A -85,B 0,C 180,E1 -30988.098,E2 -30988.098} C_VEL
LIN {X 0,Y 201.373,Z 626.103,A -85,B 0,C 180,E1 -30991.449,E2 -30991.449} C_VEL
LIN {X 0,Y 210.234,Z 628.204,A -85,B 0,C 180,E1 -30994.499,E2 -30994.499} C_VEL
LIN {X 0,Y 220.297,Z 629.154,A -85,B 0,C 180,E1 -30997.355,E2 -30997.355} C_VEL
LIN {X 0,Y 230.157,Z 628.92,A -85,B 0,C 180,E1 -30999.724,E2 -30999.724} C_VEL
LIN {X 0,Y 235.513,Z 628.378,A -85,B 0,C 180,E1 -31000.867,E2 -31000.867} C_VEL
LIN {X 0,Y 234.141,Z 629.116,A -85,B 0,C 180,E1 -31001.592,E2 -31001.592} C_VEL
LIN {X 0,Y 223.106,Z 632.374,A -85,B 0,C 180,E1 -31003.772,E2 -31003.772} C_VEL
LIN {X 0,Y 212.758,Z 634.684,A -85,B 0,C 180,E1 -31006.261,E2 -31006.261} C_VEL
LIN {X 0,Y 203.359,Z 636.101,A -85,B 0,C 180,E1 -31009.123,E2 -31009.123} C_VEL
LIN {X 0,Y 194.868,Z 636.587,A -85,B 0,C 180,E1 -31012.333,E2 -31012.333} C_VEL
LIN {X 0,Y 187.514,Z 636.268,A -85,B 0,C 180,E1 -31015.922,E2 -31015.922} C_VEL
LIN {X 0,Y 181.416,Z 635.121,A -85,B 0,C 180,E1 -31019.872,E2 -31019.872} C_VEL
LIN {X 0,Y 179.522,Z 634.504,A -85,B 0,C 180,E1 -31021.447,E2 -31021.447} C_VEL
LIN {X 0,Y 174.621,Z 640.359,A -85,B 0,C 180,E1 -31025.09,E2 -31025.09} C_VEL
LIN {X 0,Y 172.222,Z 643.339,A -85,B 0,C 180,E1 -31027.46,E2 -31027.46} C_VEL
LIN {X 0,Y 170.091,Z 645.237,A -85,B 0,C 180,E1 -31029.197,E2 -31029.197} C_VEL
LIN {X 0,Y 165.304,Z 647.693,A -85,B 0,C 180,E1 -31032.047,E2 -31032.047} C_VEL
LIN {X 0,Y 161.104,Z 649.541,A -85,B 0,C 180,E1 -31035.118,E2 -31035.118} C_VEL
LIN {X 0,Y 159.934,Z 650.447,A -85,B 0,C 180,E1 -31037.145,E2 -31037.145} C_VEL
LIN {X 0,Y 159.999,Z 652,A -85,B 0,C 180,E1 -31042.453,E2 -31042.453} C_VEL
LIN {X 0,Y 161.83,Z 652.218,A -85,B 0,C 180,E1 -31047.519,E2 -31047.519} C_VEL
LIN {X 0,Y 164.152,Z 651.858,A -85,B 0,C 180,E1 -31050.84,E2 -31050.84} C_VEL
LIN {X 0,Y 164.134,Z 659.47,A -85,B 0,C 180,E1 -31053.67,E2 -31053.67} C_VEL
LIN {X 0,Y 163.873,Z 666.607,A -85,B 0,C 180,E1 -31056.905,E2 -31056.905} C_VEL
LIN {X 0,Y 163.738,Z 675.163,A -85,B 0,C 180,E1 -31061.661,E2 -31061.661} C_VEL
LIN {X 0,Y 164.664,Z 681.802,A -85,B 0,C 180,E1 -31066.051,E2 -31066.051} C_VEL
LIN {X 0,Y 167.21,Z 688.142,A -85,B 0,C 180,E1 -31070.858,E2 -31070.858} C_VEL
LIN {X 0,Y 171.402,Z 693.428,A -85,B 0,C 180,E1 -31075.409,E2 -31075.409} C_VEL
LIN {X 0,Y 178.469,Z 698.53,A -85,B 0,C 180,E1 -31080.678,E2 -31080.678} C_VEL
LIN {X 0,Y 185.43,Z 701.526,A -85,B 0,C 180,E1 -31084.514,E2 -31084.514} C_VEL
LIN {X 0,Y 193.692,Z 703.638,A -85,B 0,C 180,E1 -31087.935,E2 -31087.935} C_VEL
LIN {X 0,Y 202.967,Z 704.769,A -85,B 0,C 180,E1 -31090.972,E2 -31090.972} C_VEL
LIN {X 0,Y 213.668,Z 704.928,A -85,B 0,C 180,E1 -31093.847,E2 -31093.847} C_VEL
LIN {X 0,Y 218.297,Z 704.679,A -85,B 0,C 180,E1 -31094.903,E2 -31094.903} C_VEL
LIN {X 0,Y 218.621,Z 704.65,A -85,B 0,C 180,E1 -31095.182,E2 -31095.182} C_VEL
LIN {X 0,Y 208.194,Z 704.924,A -85,B 0,C 180,E1 -31097.711,E2 -31097.711} C_VEL
LIN {X 0,Y 198.545,Z 704.249,A -85,B 0,C 180,E1 -31100.579,E2 -31100.579} C_VEL
LIN {X 0,Y 189.843,Z 702.599,A -85,B 0,C 180,E1 -31103.82,E2 -31103.82} C_VEL
LIN {X 0,Y 182.048,Z 699.989,A -85,B 0,C 180,E1 -31107.408,E2 -31107.408} C_VEL
LIN {X 0,Y 173.843,Z 695.193,A -85,B 0,C 180,E1 -31112.739,E2 -31112.739} C_VEL
LIN {X 0,Y 168.173,Z 689.303,A -85,B 0,C 180,E1 -31117.985,E2 -31117.985} C_VEL
LIN {X 0,Y 165.169,Z 683.212,A -85,B 0,C 180,E1 -31122.732,E2 -31122.732} C_VEL
LIN {X 0,Y 163.655,Z 675.897,A -85,B 0,C 180,E1 -31127.644,E2 -31127.644} C_VEL
LIN {X 0,Y 163.483,Z 668.137,A -85,B 0,C 180,E1 -31132.074,E2 -31132.074} C_VEL
LIN {X 0,Y 163.895,Z 660.567,A -85,B 0,C 180,E1 -31135.711,E2 -31135.711} C_VEL
LIN {X 0,Y 163.971,Z 652.678,A -85,B 0,C 180,E1 -31138.777,E2 -31138.777} C_VEL
LIN {X 0,Y 163.821,Z 642.112,A -85,B 0,C 180,E1 -31142.145,E2 -31142.145} C_VEL
LIN {X 0,Y 163.894,Z 630.466,A -85,B 0,C 180,E1 -31145.211,E2 -31145.211} C_VEL
LIN {X 0,Y 164.107,Z 618.098,A -85,B 0,C 180,E1 -31147.912,E2 -31147.912} C_VEL
LIN {X 0,Y 164.466,Z 604.233,A -85,B 0,C 180,E1 -31150.381,E2 -31150.381} C_VEL
LIN {X 0,Y 164.942,Z 589.554,A -85,B 0,C 180,E1 -31152.43,E2 -31152.43} C_VEL
LIN {X 0,Y 165.328,Z 572.38,A -85,B 0,C 180,E1 -31154.21,E2 -31154.21} C_VEL
LIN {X 0,Y 167.65,Z 481.642,A -85,B 0,C 180,E1 -31162.161,E2 -31162.161} C_VEL
LIN {X 0,Y 165.677,Z 451.682,A -85,B 0,C 180,E1 -31164.567,E2 -31164.567} C_VEL
LIN {X 0,Y 165.575,Z 439.428,A -85,B 0,C 180,E1 -31165.614,E2 -31165.614} C_VEL
LIN {X 0,Y 168.987,Z 413.211,A -85,B 0,C 180,E1 -31172.606,E2 -31172.606} C_VEL
LIN {X 0,Y 167.783,Z 406.611,A -85,B 0,C 180,E1 -31174.402,E2 -31174.402} C_VEL
LIN {X 0,Y 166.129,Z 399.329,A -85,B 0,C 180,E1 -31176.441,E2 -31176.441} C_VEL
LIN {X 0,Y 166.906,Z 401.178,A -85,B 0,C 180,E1 -31176.99,E2 -31176.99} C_VEL
LIN {X 0,Y 168.423,Z 401.69,A -85,B 0,C 180,E1 -31177.798,E2 -31177.798} C_VEL
LIN {X 0,Y 170.418,Z 400.586,A -85,B 0,C 180,E1 -31178.687,E2 -31178.687} C_VEL
LIN {X 0,Y 170.952,Z 400.098,A -85,B 0,C 180,E1 -31178.905,E2 -31178.905} C_VEL
LIN {X 0,Y 175.132,Z 399.661,A -85,B 0,C 180,E1 -31180.751,E2 -31180.751} C_VEL
LIN {X 0,Y 176.661,Z 398.853,A -85,B 0,C 180,E1 -31181.345,E2 -31181.345} C_VEL
LIN {X 0,Y 177.526,Z 399.767,A -85,B 0,C 180,E1 -31181.76,E2 -31181.76} C_VEL
LIN {X 0,Y 182.322,Z 406.745,A -85,B 0,C 180,E1 -31184.044,E2 -31184.044} C_VEL
LIN {X 0,Y 189.49,Z 418.473,A -85,B 0,C 180,E1 -31187.146,E2 -31187.146} C_VEL
LIN {X 0,Y 196.285,Z 431.417,A -85,B 0,C 180,E1 -31189.829,E2 -31189.829} C_VEL
LIN {X 0,Y 199.502,Z 438.296,A -85,B 0,C 180,E1 -31191.032,E2 -31191.032} C_VEL
LIN {X 0,Y 196.829,Z 490.384,A -85,B 0,C 180,E1 -31192.853,E2 -31192.853} C_VEL
LIN {X 0,Y 195.726,Z 504.366,A -85,B 0,C 180,E1 -31193.65,E2 -31193.65} C_VEL
LIN {X 0,Y 193.697,Z 518.657,A -85,B 0,C 180,E1 -31194.808,E2 -31194.808} C_VEL
LIN {X 0,Y 190.947,Z 532.208,A -85,B 0,C 180,E1 -31196.302,E2 -31196.302} C_VEL
LIN {X 0,Y 187.791,Z 545.061,A -85,B 0,C 180,E1 -31198.207,E2 -31198.207} C_VEL
LIN {X 0,Y 184.394,Z 556.712,A -85,B 0,C 180,E1 -31200.408,E2 -31200.408} C_VEL
LIN {X 0,Y 180.668,Z 567.396,A -85,B 0,C 180,E1 -31202.9,E2 -31202.9} C_VEL
LIN {X 0,Y 176.768,Z 577.255,A -85,B 0,C 180,E1 -31205.758,E2 -31205.758} C_VEL
LIN {X 0,Y 172.86,Z 586.689,A -85,B 0,C 180,E1 -31209.234,E2 -31209.234} C_VEL
LIN {X 0,Y 169.201,Z 595.049,A -85,B 0,C 180,E1 -31213.156,E2 -31213.156} C_VEL
LIN {X 0,Y 166.487,Z 600.92,A -85,B 0,C 180,E1 -31216.621,E2 -31216.621} C_VEL
LIN {X 0,Y 163.74,Z 607.181,A -85,B 0,C 180,E1 -31221.39,E2 -31221.39} C_VEL
LIN {X 0,Y 162.196,Z 610.812,A -85,B 0,C 180,E1 -31225.046,E2 -31225.046} C_VEL
LIN {X 0,Y 161.105,Z 614.37,A -85,B 0,C 180,E1 -31230,E2 -31230} C_VEL
LIN {X 0,Y 160.933,Z 616.576,A -85,B 0,C 180,E1 -31234.994,E2 -31234.994} C_VEL
LIN {X 0,Y 161.547,Z 617.495,A -85,B 0,C 180,E1 -31239.988,E2 -31239.988} C_VEL
LIN {X 0,Y 163.02,Z 617.132,A -85,B 0,C 180,E1 -31244.94,E2 -31244.94} C_VEL
LIN {X 0,Y 165.583,Z 615.449,A -85,B 0,C 180,E1 -31249.781,E2 -31249.781} C_VEL
LIN {X 0,Y 169.098,Z 612.409,A -85,B 0,C 180,E1 -31254.471,E2 -31254.471} C_VEL
LIN {X 0,Y 173.456,Z 607.884,A -85,B 0,C 180,E1 -31258.985,E2 -31258.985} C_VEL
LIN {X 0,Y 178.657,Z 601.732,A -85,B 0,C 180,E1 -31263.291,E2 -31263.291} C_VEL
LIN {X 0,Y 183.867,Z 594.847,A -85,B 0,C 180,E1 -31266.869,E2 -31266.869} C_VEL
LIN {X 0,Y 189.734,Z 586.266,A -85,B 0,C 180,E1 -31270.245,E2 -31270.245} C_VEL
LIN {X 0,Y 195.234,Z 577.25,A -85,B 0,C 180,E1 -31272.975,E2 -31272.975} C_VEL
LIN {X 0,Y 200.573,Z 566.786,A -85,B 0,C 180,E1 -31275.544,E2 -31275.544} C_VEL
LIN {X 0,Y 205.86,Z 555.034,A -85,B 0,C 180,E1 -31277.736,E2 -31277.736} C_VEL
LIN {X 0,Y 210.61,Z 542.532,A -85,B 0,C 180,E1 -31279.533,E2 -31279.533} C_VEL
LIN {X 0,Y 214.185,Z 530.37,A -85,B 0,C 180,E1 -31280.959,E2 -31280.959} C_VEL
LIN {X 0,Y 217.12,Z 517.458,A -85,B 0,C 180,E1 -31282.138,E2 -31282.138} C_VEL
LIN {X 0,Y 219.424,Z 503.521,A -85,B 0,C 180,E1 -31283.065,E2 -31283.065} C_VEL
LIN {X 0,Y 220.802,Z 489.767,A -85,B 0,C 180,E1 -31283.69,E2 -31283.69} C_VEL
LIN {X 0,Y 222.669,Z 460.837,A -85,B 0,C 180,E1 -31284.586,E2 -31284.586} C_VEL
LIN {X 0,Y 217.304,Z 450.18,A -85,B 0,C 180,E1 -31287.082,E2 -31287.082} C_VEL
LIN {X 0,Y 211.368,Z 439.596,A -85,B 0,C 180,E1 -31290.13,E2 -31290.13} C_VEL
LIN {X 0,Y 210.634,Z 438.406,A -85,B 0,C 180,E1 -31290.53,E2 -31290.53} C_VEL
LIN {X 0,Y 206.316,Z 451.111,A -85,B 0,C 180,E1 -31291.685,E2 -31291.685} C_VEL
LIN {X 0,Y 203.213,Z 458.53,A -85,B 0,C 180,E1 -31292.692,E2 -31292.692} C_VEL
LIN {X 0,Y 200.261,Z 463.955,A -85,B 0,C 180,E1 -31293.833,E2 -31293.833} C_VEL
LIN {X 0,Y 199.445,Z 466.543,A -85,B 0,C 180,E1 -31294.08,E2 -31294.08} C_VEL
LIN {X 0,Y 195.983,Z 478.238,A -85,B 0,C 180,E1 -31295.117,E2 -31295.117} C_VEL
LIN {X 0,Y 193.227,Z 485.843,A -85,B 0,C 180,E1 -31296.14,E2 -31296.14} C_VEL
LIN {X 0,Y 190.424,Z 491.497,A -85,B 0,C 180,E1 -31297.439,E2 -31297.439} C_VEL
LIN {X 0,Y 189.24,Z 493.608,A -85,B 0,C 180,E1 -31298.047,E2 -31298.047} C_VEL
LIN {X 0,Y 185.903,Z 504.548,A -85,B 0,C 180,E1 -31299.089,E2 -31299.089} C_VEL
LIN {X 0,Y 182.891,Z 511.81,A -85,B 0,C 180,E1 -31300.129,E2 -31300.129} C_VEL
LIN {X 0,Y 180.141,Z 516.949,A -85,B 0,C 180,E1 -31301.289,E2 -31301.289} C_VEL
LIN {X 0,Y 177.908,Z 520.175,A -85,B 0,C 180,E1 -31302.456,E2 -31302.456} C_VEL
LIN {X 0,Y 176.178,Z 522.092,A -85,B 0,C 180,E1 -31303.618,E2 -31303.618} C_VEL
LIN {X 0,Y 172.883,Z 528.277,A -85,B 0,C 180,E1 -31304.941,E2 -31304.941} C_VEL
LIN {X 0,Y 170.674,Z 531.717,A -85,B 0,C 180,E1 -31306.121,E2 -31306.121} C_VEL
LIN {X 0,Y 169.649,Z 533.083,A -85,B 0,C 180,E1 -31306.781,E2 -31306.781} C_VEL
LIN {X 0,Y 167.108,Z 535.719,A -85,B 0,C 180,E1 -31309.127,E2 -31309.127} C_VEL
LIN {X 0,Y 165.097,Z 539.196,A -85,B 0,C 180,E1 -31310.229,E2 -31310.229} C_VEL
LIN {X 0,Y 163.503,Z 541.591,A -85,B 0,C 180,E1 -31311.376,E2 -31311.376} C_VEL
LIN {X 0,Y 162.469,Z 542.862,A -85,B 0,C 180,E1 -31312.568,E2 -31312.568} C_VEL
LIN {X 0,Y 162.56,Z 541.783,A -85,B 0,C 180,E1 -31313.735,E2 -31313.735} C_VEL
